ELSE
  THIS^.stSeqCtrlGeneral.eActiveSeqState := E_SEQ_GENERAL.ERROR;
END_CASE
END_METHOD

METHOD PRIVATE _m_Seq_PRESSURE_CALIBRATION : E_SEQ_PROCESS
VAR_INPUT
END_VAR
VAR
	ActiveSeq:  STRING;
END_VAR
//THIS^._m_GeneralStepSetting(StepType:=E_STEP_STATE_TYPE.INIT,
ActiveSeq := TO_STRING(THIS^.eSeq);

CASE THIS^.stSeqCtrlGeneral.eActiveSeqState OF
E_SEQ_GENERAL.READY:;

	
E_SEQ_GENERAL.EXECUTE:;
	IF TRUE
	THEN
		THIS^.stSeqCtrlGeneral.eActiveSeqState := E_SEQ_GENERAL.RESET;
	END_IF
  
E_SEQ_GENERAL.RESET:;
	stSeqCtrlGeneral.iInternalSeqStateCase := 0;
	IF TRUE
	THEN
    THIS^.ii := 1;
    FOR THIS^.ii := 1 TO 7 BY 1 DO
      THIS^.listCalibrationTable[THIS^.ii].uiValue := 0;
      THIS^.listCalibrationTable[THIS^.ii].uiPressure := 0;
      THIS^.listCalibrationTable[THIS^.ii].uiState := 0;
		END_FOR
    THIS^.ii := 1;
		THIS^.stSeqCtrlGeneral.eActiveSeqState := E_SEQ_GENERAL.BUSY;
	END_IF
  
E_SEQ_GENERAL.BUSY:;
	CASE THIS^.stSeqCtrlGeneral.iInternalSeqStateCase OF
		0:	// Set work pressure value to XXXX
      IF TRUE
      AND THIS^.itfValve_PressureLimit.M_SetLimit(ePressureType:= E_PRESSURE_TYPE.VALUE, rLimit:= 1000 * THIS^.ii)
			THEN 
        THIS^.listCalibrationTable[THIS^.ii].uiValue := TO_UINT(1000 * THIS^.ii);
        THIS^.listCalibrationTable[THIS^.ii].uiState := 1;
        THIS^.stSeqCtrlGeneral.iInternalSeqStateCase := 10;
			END_IF
      
    10:	// Set JOG Valve off
      IF TRUE 
      AND THIS^.itfValve_AutomaticEnable.M_ToWP1(tDelay:= T#10MS)
			THEN 
        THIS^.stSeqCtrlGeneral.iInternalSeqStateCase := 20;
			END_IF
      
    20: // Set valves for WP
      IF TRUE
      AND THIS^.itfValve_SinkBlock.M_ToWP1(tDelay:= T#10MS)
      AND THIS^.itfValve_Bypass.M_ToWP1(tDelay:= T#10MS)
      AND THIS^.itfValve_CylCtrl.M_ToWP2(tDelay:= T#10MS)
      THEN
        THIS^.stSeqCtrlGeneral.iInternalSeqStateCase := 30;
			END_IF
      
    30: // Choice step
      IF TRUE
      THEN
        IF THIS^.ii = 1 THEN
          THIS^.stSeqCtrlGeneral.iInternalSeqStateCase := 40;
        ELSE
          THIS^.stSeqCtrlGeneral.iInternalSeqStateCase := 50;
				END_IF
			END_IF
      
    40: // Delay step (wait for cylinder end position)
      IF TRUE
      AND _m_Delay(DelayTime:= T#30S)
      THEN
        THIS^.stSeqCtrlGeneral.iInternalSeqStateCase := 50;
			END_IF
      
    50: // Delay step (cylinder under load)
      IF TRUE
      AND _m_Delay(DelayTime:= T#5S)
      THEN
        THIS^.stSeqCtrlGeneral.iInternalSeqStateCase := 60;
			END_IF
      
    60: // Save pressure
      IF TRUE
      THEN
        THIS^.listCalibrationTable[THIS^.ii].uiPressure := TO_UINT(THIS^.rCurrentPressureInBar);
        THIS^.listCalibrationTable[THIS^.ii].uiState := 2;
        THIS^.stSeqCtrlGeneral.iInternalSeqStateCase := 70;
			END_IF
      
    70: // Decide step
      IF TRUE
      AND _m_Delay(DelayTime:= T#1S)
      THEN
        IF THIS^.ii >= 7 OR THIS^.ii < 1 THEN
          THIS^.ii := 1;
          THIS^.stSeqCtrlGeneral.iInternalSeqStateCase := 1000;
        ELSE
          THIS^.ii := THIS^.ii + 1;
          THIS^.stSeqCtrlGeneral.iInternalSeqStateCase := 0;
				END_IF
			END_IF
      
    1000: // Stop and exit
      IF TRUE
      AND THIS^.itfValve_CylCtrl.M_ToHP(tDelay:= T#10MS)
      AND THIS^.itfValve_Bypass.M_ToHP(tDelay:= T#10MS)
			THEN 
				THIS^.stSeqCtrlGeneral.iInternalSeqStateCase := 9999;
			END_IF
      
	ELSE
		THIS^.stSeqCtrlGeneral.eActiveSeqState := E_SEQ_GENERAL.DONE;  
	END_CASE
	THIS^.stSeqCtrlGeneral.strExtraInfo := CONCAT('Internal state: ', TO_STRING(THIS^.stSeqCtrlGeneral.iInternalSeqStateCase));

E_SEQ_GENERAL.DONE:;

E_SEQ_GENERAL.ERROR:;

E_SEQ_GENERAL.TIME_OUT:; 
IF TRUE
AND THIS^.stSeqCtrlGeneral.bTimeOutActiveQuit 
THEN
  THIS^.stSeqCtrlGeneral.strExtraInfo := 'Bitte quittieren und erneut testen';
  IF TRUE
  //AND itfOpMode.P_QUIT
  THEN
    THIS^.stSeqCtrlGeneral.eActiveSeqState := E_SEQ_GENERAL.EXECUTE;
	END_IF
  
END_IF

ELSE
  THIS^.stSeqCtrlGeneral.eActiveSeqState := E_SEQ_GENERAL.ERROR;
END_CASE
END_METHOD

METHOD PRIVATE _m_Seq_SET_WORK_PRESSURE : E_SEQ_PROCESS
VAR_INPUT
END_VAR
VAR
	ActiveSeq: STRING;
END_VAR
//THIS^._m_GeneralStepSetting(StepType:=E_STEP_STATE_TYPE.INIT,
ActiveSeq := TO_STRING(THIS^.eSeq);

CASE THIS^.stSeqCtrlGeneral.eActiveSeqState OF
E_SEQ_GENERAL.READY:;

	
E_SEQ_GENERAL.EXECUTE:;
	IF TRUE
	THEN
		THIS^.stSeqCtrlGeneral.eActiveSeqState := E_SEQ_GENERAL.RESET;
	END_IF
  
E_SEQ_GENERAL.RESET:;
	stSeqCtrlGeneral.iInternalSeqStateCase := 0;
	IF TRUE
	THEN
		THIS^.stSeqCtrlGeneral.eActiveSeqState := E_SEQ_GENERAL.BUSY;
	END_IF
  
E_SEQ_GENERAL.BUSY:;
	CASE THIS^.stSeqCtrlGeneral.iInternalSeqStateCase OF
		0:	// Set work pressure
      IF TRUE
      AND THIS^.itfValve_PressureLimit.M_SetLimit(ePressureType:= E_PRESSURE_TYPE.VALUE, rLimit:= TO_REAL(THIS^.iTargetPressureAsValueA))
			THEN 
        THIS^.stSeqCtrlGeneral.iInternalSeqStateCase := 1000;
			END_IF
      
    1000: // Exit step
      IF TRUE
			THEN 
				THIS^.stSeqCtrlGeneral.iInternalSeqStateCase := 9999;
			END_IF
      
	ELSE
		THIS^.stSeqCtrlGeneral.eActiveSeqState := E_SEQ_GENERAL.DONE;  
	END_CASE
	THIS^.stSeqCtrlGeneral.strExtraInfo := CONCAT('Internal state: ', TO_STRING(THIS^.stSeqCtrlGeneral.iInternalSeqStateCase));

E_SEQ_GENERAL.DONE:;

E_SEQ_GENERAL.ERROR:;

E_SEQ_GENERAL.TIME_OUT:; 
IF TRUE
AND THIS^.stSeqCtrlGeneral.bTimeOutActiveQuit 
THEN
  THIS^.stSeqCtrlGeneral.strExtraInfo := 'Bitte quittieren und erneut testen';
  IF TRUE
  //AND itfOpMode.P_QUIT
  THEN
    THIS^.stSeqCtrlGeneral.eActiveSeqState := E_SEQ_GENERAL.EXECUTE;
	END_IF
  
END_IF

ELSE
  THIS^.stSeqCtrlGeneral.eActiveSeqState := E_SEQ_GENERAL.ERROR;
END_CASE
END_METHOD

METHOD PRIVATE _m_Seq_STOP : E_SEQ_PROCESS
VAR_INPUT
END_VAR
VAR
	ActiveSeq: STRING;
END_VAR
VAR
	
END_VAR
//THIS^._m_GeneralStepSetting(StepType:=E_STEP_STATE_TYPE.INIT,
ActiveSeq := TO_STRING(THIS^.eSeq);

CASE THIS^.stSeqCtrlGeneral.eActiveSeqState OF
E_SEQ_GENERAL.READY:;

	
E_SEQ_GENERAL.EXECUTE:;
	IF TRUE
	THEN
    THIS^.bRegulationTrigger := FALSE;
		THIS^.stSeqCtrlGeneral.eActiveSeqState := E_SEQ_GENERAL.RESET;
	END_IF
  
E_SEQ_GENERAL.RESET:;
	stSeqCtrlGeneral.iInternalSeqStateCase := 0;
	IF TRUE
	THEN
		THIS^.stSeqCtrlGeneral.eActiveSeqState := E_SEQ_GENERAL.BUSY;
	END_IF
  
E_SEQ_GENERAL.BUSY:;
	CASE THIS^.stSeqCtrlGeneral.iInternalSeqStateCase OF
		0: // Switch off valves
      IF TRUE
      AND THIS^.itfValve_Bypass.M_ToHP(tDelay:= T#0MS)
      AND THIS^.itfValve_CylCtrl.M_ToHP(tDelay:= T#0MS)
			THEN 
				THIS^.stSeqCtrlGeneral.iInternalSeqStateCase := 1000;
			END_IF
      
    1000: // Exit step
      IF TRUE
			THEN 
				THIS^.stSeqCtrlGeneral.iInternalSeqStateCase := 9999;
			END_IF
      
	ELSE
		THIS^.stSeqCtrlGeneral.eActiveSeqState := E_SEQ_GENERAL.DONE;  
	END_CASE
	THIS^.stSeqCtrlGeneral.strExtraInfo := CONCAT('Internal state: ', TO_STRING(THIS^.stSeqCtrlGeneral.iInternalSeqStateCase));

E_SEQ_GENERAL.DONE:;

E_SEQ_GENERAL.ERROR:;

E_SEQ_GENERAL.TIME_OUT:; 
IF TRUE
AND THIS^.stSeqCtrlGeneral.bTimeOutActiveQuit 
THEN
  THIS^.stSeqCtrlGeneral.strExtraInfo := 'Bitte quittieren und erneut testen';
  IF TRUE
  //AND itfOpMode.P_QUIT
  THEN
    THIS^.stSeqCtrlGeneral.eActiveSeqState := E_SEQ_GENERAL.EXECUTE;
	END_IF
  
END_IF

ELSE
  THIS^.stSeqCtrlGeneral.eActiveSeqState := E_SEQ_GENERAL.ERROR;
END_CASE
END_METHOD

METHOD PRIVATE _m_Seq_TO_HP : E_SEQ_PROCESS
VAR_INPUT
END_VAR
VAR
	ActiveSeq: STRING;
END_VAR
VAR
	
END_VAR
//THIS^._m_GeneralStepSetting(StepType:=E_STEP_STATE_TYPE.INIT,
ActiveSeq := TO_STRING(THIS^.eSeq);

CASE THIS^.stSeqCtrlGeneral.eActiveSeqState OF
E_SEQ_GENERAL.READY:;

	
E_SEQ_GENERAL.EXECUTE:;
	IF TRUE
	THEN
    THIS^.bRegulationTrigger := FALSE;
		THIS^.stSeqCtrlGeneral.eActiveSeqState := E_SEQ_GENERAL.RESET;
	END_IF
  
E_SEQ_GENERAL.RESET:;
	stSeqCtrlGeneral.iInternalSeqStateCase := 0;
	IF TRUE
	THEN
		THIS^.stSeqCtrlGeneral.eActiveSeqState := E_SEQ_GENERAL.BUSY;
	END_IF
  
E_SEQ_GENERAL.BUSY:;
	CASE THIS^.stSeqCtrlGeneral.iInternalSeqStateCase OF
		0:	// Set JOG Valve on/off
      IF TRUE 
      AND itfOpMode.P_OP_MODE_STATE = OP_MODE.AUTO
			THEN 
        IF THIS^.itfValve_AutomaticEnable.M_ToWP1(tDelay:= T#0MS) THEN
          THIS^.stSeqCtrlGeneral.iInternalSeqStateCase := 10;
				END_IF
      ELSE
        IF THIS^.itfValve_AutomaticEnable.M_ToHP(tDelay:= T#0MS) THEN
          THIS^.stSeqCtrlGeneral.iInternalSeqStateCase := 10;
				END_IF
			END_IF
      
    10:	// Set work pressure
      IF TRUE
      AND THIS^.itfValve_PressureLimit.M_SetLimit(ePressureType:= E_PRESSURE_TYPE.VALUE, rLimit:= TO_REAL(THIS^.iTargetPressureAsValueB))
			THEN 
        THIS^.stSeqCtrlGeneral.iInternalSeqStateCase := 20;
			END_IF
      
    20: // Set valves
      IF TRUE
      AND THIS^.itfValve_SinkBlock.M_ToWP1(tDelay:= T#0MS)
      AND THIS^.itfValve_Bypass.M_ToWP1(tDelay:= T#0MS)
      AND THIS^.itfValve_CylCtrl.M_ToWP1(tDelay:= T#0MS)
      THEN
        THIS^.stSeqCtrlGeneral.iInternalSeqStateCase := 1000;
			END_IF
      
    1000: // Exit step
      IF TRUE
			THEN 
				THIS^.stSeqCtrlGeneral.iInternalSeqStateCase := 9999;
			END_IF
      
	ELSE
		THIS^.stSeqCtrlGeneral.eActiveSeqState := E_SEQ_GENERAL.DONE;  
	END_CASE
	THIS^.stSeqCtrlGeneral.strExtraInfo := CONCAT('Internal state: ', TO_STRING(THIS^.stSeqCtrlGeneral.iInternalSeqStateCase));

E_SEQ_GENERAL.DONE:;
  THIS^.bRegulationTrigger := THIS^.bRegulation;

E_SEQ_GENERAL.ERROR:;

E_SEQ_GENERAL.TIME_OUT:; 
IF TRUE
AND THIS^.stSeqCtrlGeneral.bTimeOutActiveQuit 
THEN
  THIS^.stSeqCtrlGeneral.strExtraInfo := 'Bitte quittieren und erneut testen';
  IF TRUE
  //AND itfOpMode.P_QUIT
  THEN
    THIS^.stSeqCtrlGeneral.eActiveSeqState := E_SEQ_GENERAL.EXECUTE;
	END_IF
  
END_IF

ELSE
  THIS^.stSeqCtrlGeneral.eActiveSeqState := E_SEQ_GENERAL.ERROR;
END_CASE
END_METHOD

METHOD PRIVATE _m_Seq_TO_WP : E_SEQ_PROCESS
VAR_INPUT
END_VAR
VAR
	ActiveSeq: STRING;
END_VAR
VAR
	
END_VAR
//THIS^._m_GeneralStepSetting(StepType:=E_STEP_STATE_TYPE.INIT,
ActiveSeq := TO_STRING(THIS^.eSeq);

CASE THIS^.stSeqCtrlGeneral.eActiveSeqState OF
E_SEQ_GENERAL.READY:;

	
E_SEQ_GENERAL.EXECUTE:;
	IF TRUE
  //AND _m_Delay(DelayTime:= T#10MS)
	THEN
    THIS^.bRegulationTrigger := FALSE;
		THIS^.stSeqCtrlGeneral.eActiveSeqState := E_SEQ_GENERAL.RESET;
	END_IF
  
E_SEQ_GENERAL.RESET:;
	stSeqCtrlGeneral.iInternalSeqStateCase := 0;
	IF TRUE
	THEN
		THIS^.stSeqCtrlGeneral.eActiveSeqState := E_SEQ_GENERAL.BUSY;
	END_IF
  
E_SEQ_GENERAL.BUSY:;
	CASE THIS^.stSeqCtrlGeneral.iInternalSeqStateCase OF
		0:	// Set JOG Valve on/off
      IF TRUE 
      AND itfOpMode.P_OP_MODE_STATE = OP_MODE.AUTO
			THEN 
        IF THIS^.itfValve_AutomaticEnable.M_ToWP1(tDelay:= T#0MS) THEN
          THIS^.stSeqCtrlGeneral.iInternalSeqStateCase := 10;
				END_IF
      ELSE
        IF THIS^.itfValve_AutomaticEnable.M_ToHP(tDelay:= T#0MS) THEN
          THIS^.stSeqCtrlGeneral.iInternalSeqStateCase := 10;
				END_IF
			END_IF
      
    10:	// Set work pressure
      IF TRUE
      AND THIS^.itfValve_PressureLimit.M_SetLimit(ePressureType:= E_PRESSURE_TYPE.VALUE, rLimit:= TO_REAL(THIS^.iTargetPressureAsValueA))
			THEN 
        THIS^.stSeqCtrlGeneral.iInternalSeqStateCase := 20;
			END_IF
      
    20: // Valves off
      IF TRUE
      AND THIS^.itfValve_SinkBlock.M_ToWP1(tDelay:= T#0MS)
      AND THIS^.itfValve_Bypass.M_ToWP1(tDelay:= T#0MS)
      AND THIS^.itfValve_CylCtrl.M_ToWP2(tDelay:= T#0MS)
      THEN
        THIS^.stSeqCtrlGeneral.iInternalSeqStateCase := 1000;
			END_IF
      
    1000: // Exit step
      IF TRUE
			THEN 
				THIS^.stSeqCtrlGeneral.iInternalSeqStateCase := 9999;
			END_IF
      
	ELSE
		THIS^.stSeqCtrlGeneral.eActiveSeqState := E_SEQ_GENERAL.DONE;  
	END_CASE
	THIS^.stSeqCtrlGeneral.strExtraInfo := CONCAT('Internal state: ', TO_STRING(THIS^.stSeqCtrlGeneral.iInternalSeqStateCase));

E_SEQ_GENERAL.DONE:;
  THIS^.bRegulationTrigger := THIS^.bRegulation;

E_SEQ_GENERAL.ERROR:;

E_SEQ_GENERAL.TIME_OUT:; 
IF TRUE
AND THIS^.stSeqCtrlGeneral.bTimeOutActiveQuit 
THEN
  THIS^.stSeqCtrlGeneral.strExtraInfo := 'Bitte quittieren und erneut testen';
  IF TRUE
  //AND itfOpMode.P_QUIT
  THEN
    THIS^.stSeqCtrlGeneral.eActiveSeqState := E_SEQ_GENERAL.EXECUTE;
	END_IF
  
END_IF

ELSE
  THIS^.stSeqCtrlGeneral.eActiveSeqState := E_SEQ_GENERAL.ERROR;
END_CASE
END_METHOD

METHOD PRIVATE _m_SequenceManager
VAR_INPUT
END_VAR
IF FALSE
//AND THIS^.eActiveSeqState=DONE 
AND eLastSeq<>eSeq
THEN
	IF THIS^.stSeqCtrlGeneral.eActiveSeqState<>E_SEQ_GENERAL.EXECUTE THEN
		THIS^.stSeqCtrlGeneral.eActiveSeqState:=E_SEQ_GENERAL.READY;
	END_IF
END_IF

eSeq := eNextSeq;

//DelayTimer und TimeOut Timer verwalten
stSeqCtrlGeneral.bActiveStep:=	TRUE
				AND eLastSeq					=	eSeq
				AND stSeqCtrlGeneral.eLastActiveSeqState			=	stSeqCtrlGeneral.eActiveSeqState
				AND	stSeqCtrlGeneral.iLastInternalSeqStateCase	=	stSeqCtrlGeneral.iInternalSeqStateCase
				;
			
IF NOT stSeqCtrlGeneral.bActiveStep THEN
	stSeqCtrlGeneral.bDelayActive:=FALSE;
	stSeqCtrlGeneral.bTimeOutActiveQuit:=FALSE;
	stSeqCtrlGeneral.bTimeOutActiveNoQuit:=FALSE;
  THIS^.stSeqCtrlGeneral.strExtraInfo:='';
END_IF

_m_SaveLastStep();
stSeqCtrlGeneral.tonDelay	(IN:=stSeqCtrlGeneral.bActiveStep AND stSeqCtrlGeneral.bDelayActive, 		PT:=stSeqCtrlGeneral.tDelay);
stSeqCtrlGeneral.tonTimeOut	(IN:=stSeqCtrlGeneral.bActiveStep AND (stSeqCtrlGeneral.bTimeOutActiveNoQuit OR stSeqCtrlGeneral.bTimeOutActiveQuit), 	PT:=stSeqCtrlGeneral.tTimeOut);
stSeqCtrlGeneral.tonStepTime	(IN:= stSeqCtrlGeneral.bActiveStep, PT:= T#24H);

IF stSeqCtrlGeneral.tonTimeOut.Q  THEN
	stSeqCtrlGeneral.eActiveSeqState:=E_SEQ_GENERAL.TIME_OUT;
END_IF

IF stSeqCtrlGeneral.iError<>0 THEN
	eSeq:=E_SEQ_CYLINDER.ERROR_SEQ;
END_IF



eLastSeq					:=	eSeq;
stSeqCtrlGeneral.eLastActiveSeqState			:=	stSeqCtrlGeneral.eActiveSeqState;
stSeqCtrlGeneral.iLastInternalSeqStateCase	:=	stSeqCtrlGeneral.iInternalSeqStateCase;

// Reset set ready state
IF THIS^.stSeqCtrlGeneral.bExitSetReadyState THEN
  THIS^.stSeqCtrlGeneral.bExitSetReadyState := FALSE;
END_IF
END_METHOD

METHOD PRIVATE _m_TimeOut : BOOL
VAR_INPUT
	bTimeoutActiveToQuit:	BOOL;
	bTimeOutActiveNoQuit:	BOOL;
	tTimeOut:				TIME;	
END_VAR
THIS^.stSeqCtrlGeneral.bTimeOutActiveQuit:=	bTimeoutActiveToQuit;
THIS^.stSeqCtrlGeneral.bTimeOutActiveNoQuit:=	bTimeOutActiveNoQuit;
THIS^.stSeqCtrlGeneral.tTimeOut:=			tTimeOut;
_m_TimeOut:=FALSE;
IF THIS^.stSeqCtrlGeneral.tonTimeOut.Q THEN
	_m_TimeOut:=TRUE;
END_IF
END_METHOD

METHOD FB_init : BOOL
VAR_INPUT
	bInitRetains : BOOL; // if TRUE, the retain variables are initialized (warm start / cold start)
	bInCopyCode : BOOL;  // if TRUE, the instance afterwards gets moved into the copy code (online change)
  
  itfOpMode:											                        I_OP_MODE; 
  itfEventLogger:                                         I_EVENT_LOGGER;
  itfOpModeVisu:											                    I_OP_MODE_PAUSE_VISU; 
  itfValve_CylCtrl:                                       I_VALVE_X_3;
  itfValve_Bypass:                                        I_VALVE_X_2;
  itfValve_AutomaticEnable:                               I_VALVE_X_2;
  itfValve_SinkBlock:                                     I_VALVE_X_2;
  itfValve_LowPressureCircuitAdd:                         I_VALVE_X_2;
  itfValve_PressureLimit:                                 I_PRV_PROP;
  itfJogBtnPos_Pressed:                                   I_BINARY_SWITCH;
  itfJogBtnNeg_Pressed:                                   I_BINARY_SWITCH;
  lrPistonSurfaceA:                                       LREAL;
  lrPistonSurfaceB:                                       LREAL;
  rEndPosTol:                                             REAL;
  /// Volume flow in l/min or dm³/min
  rPumpVolumeFlow:                                        REAL; // Volumenstrom
  /// Pump efficiency factor (0,5-1)
  rPumpEfficiencyFactor:                                  REAL; // Wirkungsgrad
END_VAR
THIS^.itfOpMode := itfOpMode;
THIS^.itfEventLogger := itfEventLogger;
THIS^.itfOpModeVisu := itfOpModeVisu;
THIS^.itfValve_CylCtrl := itfValve_CylCtrl;
THIS^.itfValve_Bypass := itfValve_Bypass;
THIS^.itfValve_AutomaticEnable := itfValve_AutomaticEnable;
THIS^.itfValve_SinkBlock := itfValve_SinkBlock;
THIS^.itfValve_LowPressureCircuitAdd := itfValve_LowPressureCircuitAdd;
THIS^.itfValve_PressureLimit := itfValve_PressureLimit;
THIS^.itfJogBtnPos_Pressed := itfJogBtnPos_Pressed;
THIS^.itfJogBtnNeg_Pressed := itfJogBtnNeg_Pressed;
THIS^.lrPistonSurfaceA := lrPistonSurfaceA;
THIS^.lrPistonSurfaceB := lrPistonSurfaceB;
THIS^.rEndPosTol := rEndPosTol;
THIS^.rPumpVolumeFlow := rPumpVolumeFlow;
THIS^.rPumpEfficiencyFactor := rPumpEfficiencyFactor;
END_METHOD

METHOD M_AutoMode : BOOL
VAR_INPUT
	bEnable	: BOOL;
END_VAR
END_METHOD

METHOD M_LowPressureCircuit : BOOL
VAR_INPUT
  bAdd:               BOOL;
END_VAR
M_LowPressureCircuit := THIS^.stSeqCtrlGeneral.eActiveSeqState = E_SEQ_GENERAL.DONE;

// Assign input
THIS^.bLowPressureCircuitEnabled := bAdd;

// General
IF THIS^.stSeqCtrlGeneral.eActiveSeqState = E_SEQ_GENERAL.READY THEN
  THIS^.eNextSeq := E_SEQ_CYLINDER.LOW_PRESSURE_CIRCUIT;
  THIS^.stSeqCtrlGeneral.eActiveSeqState := E_SEQ_GENERAL.EXECUTE;
END_IF
END_METHOD

METHOD M_PressureCalibration : BOOL
M_PressureCalibration := THIS^.stSeqCtrlGeneral.eActiveSeqState = E_SEQ_GENERAL.DONE;

// Assign input

// General
IF THIS^.stSeqCtrlGeneral.eActiveSeqState = E_SEQ_GENERAL.READY THEN
  THIS^.eNextSeq := E_SEQ_CYLINDER.PRESSURE_CALIBRATION;
  THIS^.stSeqCtrlGeneral.eActiveSeqState := E_SEQ_GENERAL.EXECUTE;
END_IF
END_METHOD

METHOD M_Reset : BOOL
M_Reset := THIS^.stSeqCtrlGeneral.eActiveSeqState = E_SEQ_GENERAL.DONE;

// General
IF THIS^.stSeqCtrlGeneral.eActiveSeqState = E_SEQ_GENERAL.READY THEN
  THIS^.eNextSeq := E_SEQ_CYLINDER.INIT;
  THIS^.stSeqCtrlGeneral.eActiveSeqState := E_SEQ_GENERAL.EXECUTE;
END_IF
END_METHOD

{warning 'Methodenimplementierung hinzufügen'}
(*=== Method: M_Run  ============================================

 @brief: Here is the global code (Timer, Event, Flange,...)*)
METHOD M_Run
END_METHOD

METHOD M_SetReady : BOOL
VAR_INPUT
END_VAR
M_SetReady := TRUE
              AND THIS^.stSeqCtrlGeneral.eActiveSeqState = E_SEQ_GENERAL.READY
              AND THIS^.eSeq = E_SEQ_CYLINDER.BASE;

THIS^.stSeqCtrlGeneral.eActiveSeqState := E_SEQ_GENERAL.READY;
THIS^.eNextSeq := E_SEQ_CYLINDER.BASE;
END_METHOD

METHOD M_SetWorkPressure : BOOL
VAR_INPUT
  /// Bar | Force in N | Percent 0-100 | Value 0-32767
  ePressureType:                   E_PRESSURE_TYPE;
  rWorkPressure:                   REAL;
END_VAR
M_SetWorkPressure := THIS^.stSeqCtrlGeneral.eActiveSeqState = E_SEQ_GENERAL.DONE;

// Assign input
IF ePressureType = E_PRESSURE_TYPE.BAR THEN
  THIS^.rTargetPressureInBarA := THIS^.rTargetPressureInBarB := rWorkPressure;
  THIS^.rTargetPressureInForceA := rWorkPressure / 10 * THIS^.lrPistonSurfaceA;
  THIS^.rTargetPressureInForceB := rWorkPressure / 10 * THIS^.lrPistonSurfaceB;
  THIS^.rTargetPressureInPercentA := THIS^.rTargetPressureInPercentB := 100 / THIS^.itfValve_PressureLimit.P_MaxLimitInBar * rWorkPressure;
  THIS^.iTargetPressureAsValueA := THIS^.iTargetPressureAsValueB := TO_INT(F_InterpolLinear(lrValueUnscale := rWorkPressure , arrCalibrate:= listCylCalibration, iPts:= 7));
ELSIF ePressureType = E_PRESSURE_TYPE.FORCE THEN
  THIS^.rTargetPressureInForceA := THIS^.rTargetPressureInForceB := rWorkPressure;;
  THIS^.rTargetPressureInBarA := THIS^.rTargetPressureInForceA / THIS^.lrPistonSurfaceA * 10;
  THIS^.rTargetPressureInBarB := THIS^.rTargetPressureInForceB / THIS^.lrPistonSurfaceB * 10;
  THIS^.rTargetPressureInPercentA := 100 / THIS^.itfValve_PressureLimit.P_MaxLimitInBar * THIS^.rTargetPressureInBarA;
  THIS^.rTargetPressureInPercentB := 100 / THIS^.itfValve_PressureLimit.P_MaxLimitInBar * THIS^.rTargetPressureInBarB;
  THIS^.iTargetPressureAsValueA := TO_INT(F_InterpolLinear(lrValueUnscale := THIS^.rTargetPressureInBarA , arrCalibrate:= listCylCalibration, iPts:= 7));
  THIS^.iTargetPressureAsValueB := TO_INT(F_InterpolLinear(lrValueUnscale := THIS^.rTargetPressureInBarB , arrCalibrate:= listCylCalibration, iPts:= 7));
ELSIF ePressureType = E_PRESSURE_TYPE.PERCENT THEN
  THIS^.rTargetPressureInPercentA := THIS^.rTargetPressureInPercentB := rWorkPressure;
  THIS^.rTargetPressureInBarA := THIS^.rTargetPressureInBarB := THIS^.itfValve_PressureLimit.P_MaxLimitInBar / 100 * rWorkPressure;
  THIS^.rTargetPressureInForceA := THIS^.rTargetPressureInBarA / 10 * THIS^.lrPistonSurfaceA;
  THIS^.rTargetPressureInForceB := THIS^.rTargetPressureInBarB / 10 * THIS^.lrPistonSurfaceB;
  THIS^.iTargetPressureAsValueA := TO_INT(F_InterpolLinear(lrValueUnscale := THIS^.rTargetPressureInBarA , arrCalibrate:= listCylCalibration, iPts:= 7));
  THIS^.iTargetPressureAsValueB := TO_INT(F_InterpolLinear(lrValueUnscale := THIS^.rTargetPressureInBarB , arrCalibrate:= listCylCalibration, iPts:= 7));
ELSE
  THIS^.iTargetPressureAsValueA := THIS^.iTargetPressureAsValueB := TO_INT(rWorkPressure);
END_IF

// General
IF THIS^.stSeqCtrlGeneral.eActiveSeqState = E_SEQ_GENERAL.READY THEN
  THIS^.eNextSeq := E_SEQ_CYLINDER.SET_WORK_PRESSURE;
  THIS^.stSeqCtrlGeneral.eActiveSeqState := E_SEQ_GENERAL.EXECUTE;
END_IF
END_METHOD

METHOD M_SetWorkPressureZero : BOOL
M_SetWorkPressureZero := THIS^.stSeqCtrlGeneral.eActiveSeqState = E_SEQ_GENERAL.DONE;

THIS^.iTargetPressureAsValueA := 0;

// General
IF THIS^.stSeqCtrlGeneral.eActiveSeqState = E_SEQ_GENERAL.READY THEN
  THIS^.eNextSeq := E_SEQ_CYLINDER.SET_WORK_PRESSURE;
  THIS^.stSeqCtrlGeneral.eActiveSeqState := E_SEQ_GENERAL.EXECUTE;
END_IF
END_METHOD

METHOD M_Stop : BOOL
M_Stop := THIS^.stSeqCtrlGeneral.eActiveSeqState = E_SEQ_GENERAL.DONE;

// Assign input
THIS^.bRegulation := FALSE;
THIS^.rActiveForce := 0;
THIS^.iCorrectedPressureAsValue := 0;
THIS^.bRegulationTrigger := FALSE;
THIS^.bRegulationBusy := FALSE;
THIS^.bCorrectionTrigger := FALSE;

// General
IF THIS^.stSeqCtrlGeneral.eActiveSeqState = E_SEQ_GENERAL.READY THEN
  THIS^.eNextSeq := E_SEQ_CYLINDER.STOP;
  THIS^.stSeqCtrlGeneral.eActiveSeqState := E_SEQ_GENERAL.EXECUTE;
END_IF
END_METHOD

METHOD M_ToHP : BOOL
VAR_INPUT
  /// Bar | Force in N | Percent 0-100 | Value 0-32767
  ePressureType:            E_PRESSURE_TYPE;
  rWorkPressure:            REAL;
  bPressureRegulation:      BOOL;
  /// Just need for prop valve
  eSpeedType:               E_SPEED_TYPE;
  rSpeed:                   REAL; 
END_VAR
M_ToHP := THIS^.stSeqCtrlGeneral.eActiveSeqState = E_SEQ_GENERAL.DONE;

// Assign input
IF ePressureType = E_PRESSURE_TYPE.BAR THEN
  THIS^.rTargetPressureInBarA := THIS^.rTargetPressureInBarB := rWorkPressure;
  THIS^.rTargetPressureInForceA := rWorkPressure / 10 * THIS^.lrPistonSurfaceA;
  THIS^.rTargetPressureInForceB := rWorkPressure / 10 * THIS^.lrPistonSurfaceB;
  THIS^.rTargetPressureInPercentA := THIS^.rTargetPressureInPercentB := 100 / THIS^.itfValve_PressureLimit.P_MaxLimitInBar * rWorkPressure;
  THIS^.iTargetPressureAsValueA := THIS^.iTargetPressureAsValueB := THIS^.iCorrectedPressureAsValue := TO_INT(F_InterpolLinear(lrValueUnscale := rWorkPressure , arrCalibrate:= listCylCalibration, iPts:= 7));
ELSIF ePressureType = E_PRESSURE_TYPE.FORCE THEN
  THIS^.rTargetPressureInForceA := THIS^.rTargetPressureInForceB := rWorkPressure;;
  THIS^.rTargetPressureInBarA := THIS^.rTargetPressureInForceA / THIS^.lrPistonSurfaceA * 10;
  THIS^.rTargetPressureInBarB := THIS^.rTargetPressureInForceB / THIS^.lrPistonSurfaceB * 10;
  THIS^.rTargetPressureInPercentA := 100 / THIS^.itfValve_PressureLimit.P_MaxLimitInBar * THIS^.rTargetPressureInBarA;
  THIS^.rTargetPressureInPercentB := 100 / THIS^.itfValve_PressureLimit.P_MaxLimitInBar * THIS^.rTargetPressureInBarB;
  THIS^.iTargetPressureAsValueA := THIS^.iCorrectedPressureAsValue := TO_INT(F_InterpolLinear(lrValueUnscale := THIS^.rTargetPressureInBarA , arrCalibrate:= listCylCalibration, iPts:= 7));
  THIS^.iTargetPressureAsValueB := TO_INT(F_InterpolLinear(lrValueUnscale := THIS^.rTargetPressureInBarB , arrCalibrate:= listCylCalibration, iPts:= 7));
ELSIF ePressureType = E_PRESSURE_TYPE.PERCENT THEN
  THIS^.rTargetPressureInPercentA := THIS^.rTargetPressureInPercentB := rWorkPressure;
  THIS^.rTargetPressureInBarA := THIS^.rTargetPressureInBarB := THIS^.itfValve_PressureLimit.P_MaxLimitInBar / 100 * rWorkPressure;
  THIS^.rTargetPressureInForceA := THIS^.rTargetPressureInBarA / 10 * THIS^.lrPistonSurfaceA;
  THIS^.rTargetPressureInForceB := THIS^.rTargetPressureInBarB / 10 * THIS^.lrPistonSurfaceB;
  THIS^.iTargetPressureAsValueA := THIS^.iCorrectedPressureAsValue := TO_INT(F_InterpolLinear(lrValueUnscale := THIS^.rTargetPressureInBarA , arrCalibrate:= listCylCalibration, iPts:= 7));
  THIS^.iTargetPressureAsValueB := TO_INT(F_InterpolLinear(lrValueUnscale := THIS^.rTargetPressureInBarB , arrCalibrate:= listCylCalibration, iPts:= 7));
ELSE
  THIS^.iTargetPressureAsValueA := THIS^.iTargetPressureAsValueB := THIS^.iCorrectedPressureAsValue := TO_INT(rWorkPressure);
END_IF
THIS^.bRegulation := bPressureRegulation;

// General
IF THIS^.stSeqCtrlGeneral.eActiveSeqState = E_SEQ_GENERAL.READY THEN
  THIS^.eNextSeq := E_SEQ_CYLINDER.TO_HP;
  THIS^.stSeqCtrlGeneral.eActiveSeqState := E_SEQ_GENERAL.EXECUTE;
END_IF
END_METHOD

METHOD M_ToWP : BOOL
VAR_INPUT
  /// Bar | Force in N | Percent 0-100 | Value 0-32767
  ePressureType:            E_PRESSURE_TYPE;
  rWorkPressure:            REAL;
  bPressureRegulation:      BOOL;
  /// Just need for prop valve
  eSpeedType:               E_SPEED_TYPE;
  rSpeed:                   REAL; 
END_VAR
M_ToWP := THIS^.stSeqCtrlGeneral.eActiveSeqState = E_SEQ_GENERAL.DONE;

// Assign input
IF ePressureType = E_PRESSURE_TYPE.BAR THEN
  THIS^.rTargetPressureInBarA := THIS^.rTargetPressureInBarB := rWorkPressure;
  THIS^.rTargetPressureInForceA := rWorkPressure / 10 * THIS^.lrPistonSurfaceA;
  THIS^.rTargetPressureInForceB := rWorkPressure / 10 * THIS^.lrPistonSurfaceB;
  THIS^.rTargetPressureInPercentA := THIS^.rTargetPressureInPercentB := 100 / THIS^.itfValve_PressureLimit.P_MaxLimitInBar * rWorkPressure;
  THIS^.iTargetPressureAsValueA := THIS^.iTargetPressureAsValueB := THIS^.iCorrectedPressureAsValue := TO_INT(F_InterpolLinear(lrValueUnscale := rWorkPressure , arrCalibrate:= listCylCalibration, iPts:= 7));
ELSIF ePressureType = E_PRESSURE_TYPE.FORCE THEN
  THIS^.rTargetPressureInForceA := THIS^.rTargetPressureInForceB := rWorkPressure;;
  THIS^.rTargetPressureInBarA := THIS^.rTargetPressureInForceA / THIS^.lrPistonSurfaceA * 10;
  THIS^.rTargetPressureInBarB := THIS^.rTargetPressureInForceB / THIS^.lrPistonSurfaceB * 10;
  THIS^.rTargetPressureInPercentA := 100 / THIS^.itfValve_PressureLimit.P_MaxLimitInBar * THIS^.rTargetPressureInBarA;
  THIS^.rTargetPressureInPercentB := 100 / THIS^.itfValve_PressureLimit.P_MaxLimitInBar * THIS^.rTargetPressureInBarB;
  THIS^.iTargetPressureAsValueA := THIS^.iCorrectedPressureAsValue := TO_INT(F_InterpolLinear(lrValueUnscale := THIS^.rTargetPressureInBarA , arrCalibrate:= listCylCalibration, iPts:= 7));
  THIS^.iTargetPressureAsValueB := TO_INT(F_InterpolLinear(lrValueUnscale := THIS^.rTargetPressureInBarB , arrCalibrate:= listCylCalibration, iPts:= 7));
ELSIF ePressureType = E_PRESSURE_TYPE.PERCENT THEN
  THIS^.rTargetPressureInPercentA := THIS^.rTargetPressureInPercentB := rWorkPressure;
  THIS^.rTargetPressureInBarA := THIS^.rTargetPressureInBarB := THIS^.itfValve_PressureLimit.P_MaxLimitInBar / 100 * rWorkPressure;
  THIS^.rTargetPressureInForceA := THIS^.rTargetPressureInBarA / 10 * THIS^.lrPistonSurfaceA;
  THIS^.rTargetPressureInForceB := THIS^.rTargetPressureInBarB / 10 * THIS^.lrPistonSurfaceB;
  THIS^.iTargetPressureAsValueA := THIS^.iCorrectedPressureAsValue := TO_INT(F_InterpolLinear(lrValueUnscale := THIS^.rTargetPressureInBarA , arrCalibrate:= listCylCalibration, iPts:= 7));
  THIS^.iTargetPressureAsValueB := TO_INT(F_InterpolLinear(lrValueUnscale := THIS^.rTargetPressureInBarB , arrCalibrate:= listCylCalibration, iPts:= 7));
ELSE
  THIS^.iTargetPressureAsValueA := THIS^.iTargetPressureAsValueB := THIS^.iCorrectedPressureAsValue := TO_INT(rWorkPressure);
END_IF
THIS^.bRegulation := bPressureRegulation;

// General
IF THIS^.stSeqCtrlGeneral.eActiveSeqState = E_SEQ_GENERAL.READY THEN
  THIS^.eNextSeq := E_SEQ_CYLINDER.TO_WP;
  THIS^.stSeqCtrlGeneral.eActiveSeqState := E_SEQ_GENERAL.EXECUTE;
END_IF
END_METHOD

{warning 'Eigenschaftenimplementierung hinzufügen'}
PROPERTY P_CurrentForceInKN : REAL
GET
IF THIS^.itfValve_CylCtrl.P_InWP2 THEN
  P_CurrentForceInKN := THIS^.rCurrentPressureInBar / 10000 * THIS^.lrPistonSurfaceA;
  THIS^.rActiveForce := THIS^.rTargetPressureInForceA;
ELSIF THIS^.itfValve_CylCtrl.P_InWP1 THEN
  P_CurrentForceInKN := THIS^.rCurrentPressureInBar / 10000 * THIS^.lrPistonSurfaceB;
  THIS^.rActiveForce := THIS^.rTargetPressureInForceB;
ELSE
  P_CurrentForceInKN := 0;
END_IF
END_GET
END_PROPERTY

{warning 'Eigenschaftenimplementierung hinzufügen'}
(*=== Property: P_Event  ============================================

 @param [set]: 	Set the Structure "ST_EVENT" from another Object
 @param [get]: 	Return the Structure "ST_EVENT", it contains the actual 
					event of the Object *)
PROPERTY P_Event : GenLib.ST_EVENT
GET
END_GET
SET
END_SET
END_PROPERTY

{warning 'Eigenschaftenimplementierung hinzufügen'}
(*=== Property: P_FullObjectPath  ============================================

 @param [set]: 	Set the Object Path (Clear String of Object)
 @param [get]: 	Return the Objectpath *)
PROPERTY P_FullObjectPath : STRING
GET
P_FullObjectPath := strInstancePath;
END_GET
SET
strInstancePath := P_FullObjectPath;
END_SET
END_PROPERTY

{warning 'Eigenschaftenimplementierung hinzufügen'}
(*=== Property: P_Global_Ack  ============================================

 @param [set]: 	Set the Bit for Ack from another Object
 @param [get]: 	Return the state of Ack Bit*)
PROPERTY P_Global_Ack : BOOL
GET
END_GET
SET
END_SET
END_PROPERTY

{warning 'Eigenschaftenimplementierung hinzufügen'}
(*=== Property: P_GlobalID  ============================================

 @param [set]: 	-
 @param [get]: 	Return the string of instance path*)
PROPERTY P_GlobalID : STRING
GET
END_GET
END_PROPERTY

{warning 'Eigenschaftenimplementierung hinzufügen'}
PROPERTY P_PistonSurfaceA : LREAL
GET
P_PistonSurfaceA := THIS^.lrPistonSurfaceA;
END_GET
END_PROPERTY

{warning 'Eigenschaftenimplementierung hinzufügen'}
PROPERTY P_PistonSurfaceB : LREAL
GET
P_PistonSurfaceB := THIS^.lrPistonSurfaceB;
END_GET
END_PROPERTY

{warning 'Eigenschaftenimplementierung hinzufügen'}
PROPERTY P_PressureOk : BOOL
GET
END_GET
END_PROPERTY

{warning 'Eigenschaftenimplementierung hinzufügen'}
PROPERTY P_ReadyState : BOOL
GET
P_ReadyState := THIS^.stSeqCtrlGeneral.eActiveSeqState = E_SEQ_GENERAL.READY;
END_GET
END_PROPERTY

PROPERTY P_WorkPressure : REAL
GET
P_WorkPressure := THIS^.rCurrentPressureInBar;
END_GET
END_PROPERTY

END_FUNCTION_BLOCK

// ---- PROGRAMS/PrgVisu.TcPOU
{attribute 'global_init_slot' := '40030'}
PROGRAM PrgVisu
VAR
	fbVisuOPMode:						                        FB_OP_MODE_PAUSE_VISU(itfOpMode:= PrgOrg.fbOpMode);
  tonHeartbeat:                                   TON;
  
  bInit : 									                      BOOL; 
  bSend : 									                      BOOL; 
  fbMsg : 									                      FB_TcMessage;
  fbAlarm:                                        FB_TcAlarm;
  bMachineLightOn:                                BOOL := TRUE;
  fbEventLogger:                                  FB_EVENT_LOGGER();
END_VAR
VAR //HMI enables
  fbHMICtrl:                                      FB_HMI_CTRL_ADS(itfOpMode:= PrgOrg.fbOpMode,
                                                                  itfEventLogger:= PrgOrg.fbEventLogger);
  bEnableAuto:                                    BOOL;
  bEnableEnduranceRun:                            BOOL;
  bEnableLeakTest1:                               BOOL;
  bEnableLeakTest2:                               BOOL;
  bEnableBreakPressureDet:                        BOOL;
  bEnableManual:                                  BOOL;
  bEnableHand:                                    BOOL;
  bEnableJog:                                     BOOL;
  bEnableInit:                                    BOOL;
  bEnableDoorLock:                                BOOL;
  bEnableAck:                                     BOOL;
  bEnableParams:                                  BOOL;
  bEnableOptions:                                 BOOL;
  bEnableSelection:                               BOOL;
  bPumpsOn:                                       BOOL;
END_VAR
VAR
  uiHMISeq:                                       UINT := 0;
  bStartHMI:                                      BOOL;
  bCloseHMI:                                      BOOL;
  bOpenKeyboard:                                  BOOL;
  bHideKeyboard:                                  BOOL;
  bShutdownPc:                                    BOOL;
  bRestartPc:                                     BOOL;
  liFreeSpaceOnC:                                 LINT;
END_VAR
VAR // Parameter: Selected ComboBox Index
  uiCmbCylinder:                                  UINT := 0;
  uiCmbEnduranceRun:                              UINT := 0;
  uiCmbGeneralSettings:                           UINT := 0;
  uiCmbLeakTest1:                                 UINT := 0;
  uiCmbLeakTest2:                                 UINT := 0;
  uiCmbBreakPressureDet:                          UINT := 0;
END_VAR

(* Actions *)
A_000_FBs();
A_010_Init();
A_020_Enables();
A_030_HMIControl();

ACTION A_000_FBs:
(* FBs *)
fbVisuOPMode();
fbHMICtrl(bLifeBit:= PrgMeasure.bLifeBit,
          bAdsConnected:= PrgMeasure.bAdsConnected,
          bReady:= PrgMeasure.bReady,
          bBusy:= PrgMeasure.bBusy,
          liFreeSpaceOnC=> liFreeSpaceOnC);
END_ACTION

ACTION A_010_Init:
tonHeartbeat(in:=NOT tonHeartbeat.Q, pt:=T#100MS);
END_ACTION

ACTION A_020_Enables:
(* Enables *)
bPumpsOn := TRUE
            AND PrgStation.fbBypassPump.P_State
            AND PrgStation.fbCounterCyl1Pump.P_State
            AND PrgStation.fbCounterCyl2Pump.P_State
            AND PrgStation.fbCounterCyl3Pump.P_State
            AND PrgStation.fbCounterCyl4Pump.P_State
            AND PrgStation.fbLowPressurePump.P_State
            AND PrgStation.fbOilCooler.P_State
            AND PrgStation.fbTestCyl1Pump.P_State
            AND PrgStation.fbTestCyl2Pump.P_State
            AND PrgStation.fbTestCyl3Pump.P_State
            AND PrgStation.fbTestCyl4Pump.P_State;
            
bEnableAuto := TRUE
               AND (bEnableEnduranceRun
                 OR bEnableLeakTest1
                 OR bEnableLeakTest2
                 OR bEnableBreakPressureDet);

bEnableEnduranceRun := TRUE
               AND (NOT (fbVisuOPMode.b_Automatic OR fbVisuOPMode.b_Manual OR fbVisuOPMode.b_Reset)
               AND PrgOrg.bInitOK
               AND ((PrgStation.fbNest1.bEnable AND PrgStation.sTestCyl1SNo<>'') 
                 OR (PrgStation.fbNest2.bEnable AND PrgStation.sTestCyl2SNo<>'') 
                 OR (PrgStation.fbNest3.bEnable AND PrgStation.sTestCyl2SNo<>'')
                 OR (PrgStation.fbNest4.bEnable AND PrgStation.sTestCyl2SNo<>''))
               AND NOT PrgOrg.fbOpMode.P_EMERGANCY_STOP
               AND bPumpsOn
               AND PrgOrg.fbFromSafety_SafetyDoor_Ok.P_Active);
               
bEnableLeakTest1 := TRUE
                    AND (NOT (fbVisuOPMode.b_Automatic OR fbVisuOPMode.b_Manual OR fbVisuOPMode.b_Reset)
                    AND PrgOrg.bInitOK
                    AND ((PrgStation.fbNest1.bEnable AND PrgStation.sTestCyl1SNo<>'') 
                      OR (PrgStation.fbNest2.bEnable AND PrgStation.sTestCyl2SNo<>'') 
                      OR (PrgStation.fbNest3.bEnable AND PrgStation.sTestCyl2SNo<>'')
                      OR (PrgStation.fbNest4.bEnable AND PrgStation.sTestCyl2SNo<>''))
                    AND NOT PrgOrg.fbOpMode.P_EMERGANCY_STOP
                    AND bPumpsOn
                    AND PrgOrg.fbFromSafety_SafetyDoor_Ok.P_Active);
                    
bEnableLeakTest2 := TRUE
                    AND (NOT (fbVisuOPMode.b_Automatic OR fbVisuOPMode.b_Manual OR fbVisuOPMode.b_Reset)
                    AND PrgOrg.bInitOK
                    AND (PrgStation.fbNest1.bEnable AND PrgStation.sTestCyl1SNo<>'')
                    AND NOT PrgOrg.fbOpMode.P_EMERGANCY_STOP
                    AND bPumpsOn
                    AND PrgOrg.fbFromSafety_SafetyDoor_Ok.P_Active);
                    
bEnableBreakPressureDet := TRUE
                           AND (NOT (fbVisuOPMode.b_Automatic OR fbVisuOPMode.b_Manual OR fbVisuOPMode.b_Reset)
                           AND PrgOrg.bInitOK
                           AND (PrgStation.fbNest1.bEnable AND PrgStation.sTestCyl1SNo<>'')
                           AND NOT PrgOrg.fbOpMode.P_EMERGANCY_STOP
                           AND bPumpsOn
                           AND PrgOrg.fbFromSafety_SafetyDoor_Ok.P_Active);
               
bEnableManual := TRUE
                 AND (bEnableHand
                   OR bEnableJog);
               
bEnableHand := TRUE
               AND (NOT (fbVisuOPMode.b_Automatic 
                 OR fbVisuOPMode.b_Manual 
                 OR fbVisuOPMode.b_Reset) 
               AND bPumpsOn
               AND PrgOrg.fbFromSafety_SafetyDoor_Ok.P_Active);
                 
bEnableJog := TRUE
              AND (NOT (fbVisuOPMode.b_Automatic 
                OR fbVisuOPMode.b_Manual 
                OR fbVisuOPMode.b_Reset) 
              AND bPumpsOn);
                 
bEnableInit := TRUE
               AND (NOT (fbVisuOPMode.b_Automatic 
                 OR fbVisuOPMode.b_Manual 
                 OR fbVisuOPMode.b_Reset 
                 OR PrgStation.bBusyInit)
               AND PrgOrg.fbFromSafety_SafetyDoor_Ok.P_Active);
                 
bEnableDoorLock := TRUE
                   AND (NOT (fbVisuOPMode.b_Automatic 
                     OR fbVisuOPMode.b_Reset) 
                   OR PrgStation.fbMainProcess.bShowMessage);
                   
bEnableAck := TRUE
              AND (NOT (fbVisuOPMode.b_Automatic 
                OR fbVisuOPMode.b_Reset));
                
bEnableParams := TRUE
                 AND PrgOrg.fbOpMode.P_OP_MODE_STATE = OP_MODE.AUTO_TEMPORARY;
                 
bEnableSelection := TRUE
                    AND NOT fbVisuOPMode.b_Automatic;
                 
bEnableOptions := TRUE
                  AND (NOT (fbVisuOPMode.b_Automatic 
                   OR fbVisuOPMode.b_Reset));
END_ACTION

ACTION A_030_HMIControl:
(* HMI control *)
CASE uiHMISeq OF
  0:
    IF fbHMICtrl.M_SetReady() THEN
      IF bStartHMI THEN
        uiHMISeq := 1;
      ELSIF bCloseHMI THEN
        uiHMISeq := 2;
      ELSIF bOpenKeyboard THEN
        uiHMISeq := 3;
      ELSIF bHideKeyboard THEN
        uiHMISeq := 4;
      ELSIF bShutdownPc THEN
        uiHMISeq := 5;
      ELSIF bRestartPc THEN
        uiHMISeq := 6;
			END_IF
		END_IF
  1:
    IF fbHMICtrl.M_StartHMI() THEN
      bStartHMI := FALSE;
      uiHMISeq := 0;
		END_IF
  2:
    IF fbHMICtrl.M_CloseHMI() THEN
      bCloseHMI := FALSE;
      uiHMISeq := 0;
		END_IF
  3:
    IF fbHMICtrl.M_ShowWinKeyboard() THEN
      bOpenKeyboard := FALSE;
      uiHMISeq := 0;
		END_IF
  4:
    IF fbHMICtrl.M_HideWinKeyboard() THEN
      bHideKeyboard := FALSE;
      uiHMISeq := 0;
		END_IF
  5:
    IF fbHMICtrl.M_PCShutdown() THEN
      bShutdownPc := FALSE;
      uiHMISeq := 0;
		END_IF
  6:
    IF fbHMICtrl.M_PCReboot() THEN
      bRestartPc := FALSE;
      uiHMISeq := 0;
		END_IF
END_CASE
END_ACTION

END_PROGRAM

// ---- ORGANISATION/OP_MODE/POU/FB_OP_MODE_PAUSE_VISU.TcPOU
FUNCTION_BLOCK FB_OP_MODE_PAUSE_VISU IMPLEMENTS I_OP_MODE_PAUSE_VISU
VAR
	itfOpMode:                          I_OP_MODE_PAUSE;
	//Press 
	bClick_Automatic:                   BOOL;
	bClick_Debug:                       BOOL;
	bClick_Manual:                      BOOL;
	bClick_Reset:                       BOOL;
	bClick_Start:                       BOOL;
	bClick_Stop:                        BOOL;
	bClick_Pause:                       BOOL;
	//State
	b_Automatic:                        BOOL;
	b_Debug:                            BOOL;
	b_Manual:                           BOOL;
	b_Reset:                            BOOL;
	//temporay State
	btemporay_Automatic:                BOOL;
	btemporay_Debug:                    BOOL;
	btemporay_Manual:                   BOOL;
	btemporay_Reset:                    BOOL;
	iOPModeState:                       INT;
  // Control buttons clicked
  bEnduranceRunClicked:               BOOL;
  bLeakTest1Clicked:                  BOOL;
  bLeakTest2Clicked:                  BOOL;
  bBreakTestClicked:                  BOOL;
  bJogClicked:                        BOOL;
  bHandClicked:                       BOOL;
  bEnduranceRunMode:                  BOOL;
  bLeakTest1Mode:                     BOOL;
  bLeakTest2Mode:                     BOOL;
  bBreakTestMode:                     BOOL;
  bJogMode:                           BOOL;
  bHandMode:                          BOOL;
  
  // JOG Direction
  bJogCounterCyl1_Clicked:            BOOL;
  bJogCounterCyl2_Clicked:            BOOL;
  bJogCounterCyl3_Clicked:            BOOL;
  bJogCounterCyl4_Clicked:            BOOL;
  bJogCounterCyl1_Active:             BOOL;
  bJogCounterCyl2_Active:             BOOL;
  bJogCounterCyl3_Active:             BOOL;
  bJogCounterCyl4_Active:             BOOL;
	fbBlink:                            FB_Blink;
END_VAR
VAR_IN_OUT

END_VAR
VAR
END_VAR


//CLICK to OP-Mode
IF bClick_Automatic	THEN
	itfOpMode.M_AUTOMATIC();
	bClick_Automatic := FALSE;
END_IF
	
IF bClick_Debug	THEN
	itfOpMode.M_DEBUG();
	bClick_Debug := FALSE;
END_IF
		
IF bClick_Manual THEN
	itfOpMode.M_MANUAL();
	bClick_Manual		:= FALSE;
END_IF
			
IF bClick_Reset	THEN
	itfOpMode.M_RESET();
	bClick_Reset		:= FALSE;
  //M_ResetModeSelection();
END_IF
	
		
IF bClick_Start	THEN
	itfOpMode.M_OP_MODE_ON();
	bClick_Start := FALSE;
END_IF
		
IF bClick_Stop THEN
	itfOpMode.M_OP_MODE_OFF();
  //itfOpMode.M_STOP();
	bClick_Stop			:= FALSE;
  //M_ResetModeSelection();
END_IF

IF bClick_Pause	THEN
	itfOpMode.M_OP_MODE_TO_PAUSE();
	bClick_Pause := FALSE;
END_IF
//
b_Automatic := FALSE;
b_Debug := FALSE; 
b_Manual := FALSE;
b_Reset := FALSE;
btemporay_Automatic := FALSE;
btemporay_Debug := FALSE;
btemporay_Manual := FALSE;
btemporay_Reset := FALSE;

//GET OP MODE STATE
CASE itfOpMode.P_OP_MODE_STATE OF		
	OP_MODE.AUTO: 				    b_Automatic := TRUE;
	OP_MODE.PAUSE:				    b_Automatic :=fbBlink.P_1Hz;		
 	OP_MODE.DEBUG:				    b_Debug := TRUE;
	OP_MODE.MANUAL:				    b_Manual := TRUE;
	OP_MODE.INIT:				      b_Reset := fbBlink.P_1Hz;
	OP_MODE.INIT_OK:			    b_Reset := TRUE;							
	OP_MODE.AUTO_TEMPORARY:		btemporay_Automatic := TRUE;
	OP_MODE.DEBUG_TEMPORARY:	btemporay_Debug := TRUE;
	OP_MODE.MANUAL_TEMPORARY:	btemporay_Manual := TRUE;
	OP_MODE.RESET_TEMPORARY:	btemporay_Reset := TRUE;
END_CASE
iOPModeState := itfOpMode.P_OP_MODE_STATE;

// Control buttons clicked
IF bEnduranceRunClicked THEN
  bEnduranceRunClicked := FALSE;
  bEnduranceRunMode := TRUE;
  bLeakTest1Mode := FALSE;
  bLeakTest2Mode := FALSE;
  bBreakTestMode := FALSE;
  bJogMode := FALSE;
  bHandMode := FALSE;
ELSIF bLeakTest1Clicked THEN
  bLeakTest1Clicked := FALSE;
  bEnduranceRunMode := FALSE;
  bLeakTest1Mode := TRUE;
  bLeakTest2Mode := FALSE;
  bBreakTestMode := FALSE;
  bJogMode := FALSE;
  bHandMode := FALSE;
ELSIF bLeakTest2Clicked THEN
  bLeakTest2Clicked := FALSE;
  bEnduranceRunMode := FALSE;
  bLeakTest1Mode := FALSE;
  bLeakTest2Mode := TRUE;
  bBreakTestMode := FALSE;
  bJogMode := FALSE;
  bHandMode := FALSE;
ELSIF bBreakTestClicked THEN
  bBreakTestClicked := FALSE;
  bEnduranceRunMode := FALSE;
  bLeakTest1Mode := FALSE;
  bLeakTest2Mode := FALSE;
  bBreakTestMode := TRUE;
  bJogMode := FALSE;
  bHandMode := FALSE;
ELSIF bJogClicked THEN
  bJogClicked := FALSE;
  bEnduranceRunMode := FALSE;
  bLeakTest1Mode := FALSE;
  bLeakTest2Mode := FALSE;
  bBreakTestMode := FALSE;
  bJogMode := TRUE;
  bHandMode := FALSE;
ELSIF bHandClicked THEN
  bHandClicked := FALSE;
  bEnduranceRunMode := FALSE;
  bLeakTest1Mode := FALSE;
  bLeakTest2Mode := FALSE;
  bBreakTestMode := FALSE;
  bJogMode := FALSE;
  bHandMode := TRUE;
END_IF

IF bJogCounterCyl1_Clicked THEN
  bJogCounterCyl1_Clicked := FALSE;
  bJogCounterCyl1_Active := TRUE;
  bJogCounterCyl2_Active := FALSE;
  bJogCounterCyl3_Active := FALSE;
  bJogCounterCyl4_Active := FALSE;
ELSIF bJogCounterCyl2_Clicked THEN
  bJogCounterCyl2_Clicked := FALSE;
  bJogCounterCyl1_Active := FALSE;
  bJogCounterCyl2_Active := TRUE;
  bJogCounterCyl3_Active := FALSE;
  bJogCounterCyl4_Active := FALSE;
ELSIF bJogCounterCyl3_Clicked THEN
  bJogCounterCyl3_Clicked := FALSE;
  bJogCounterCyl1_Active := FALSE;
  bJogCounterCyl2_Active := FALSE;
  bJogCounterCyl3_Active := TRUE;
  bJogCounterCyl4_Active := FALSE;
ELSIF bJogCounterCyl4_Clicked THEN
  bJogCounterCyl4_Clicked := FALSE;
  bJogCounterCyl1_Active := FALSE;
  bJogCounterCyl2_Active := FALSE;
  bJogCounterCyl3_Active := FALSE;
  bJogCounterCyl4_Active := TRUE;
END_IF

METHOD FB_init : BOOL
VAR_INPUT
	bInitRetains : BOOL; // if TRUE, the retain variables are initialized (warm start / cold start)
	bInCopyCode : BOOL;  // if TRUE, the instance afterwards gets moved into the copy code (online change)
  
	itfOpMode:  I_OP_MODE_PAUSE;
END_VAR
THIS^.itfOpMode := itfOpMode;
END_METHOD

METHOD M_ResetModeSelection : BOOL
VAR_INPUT
END_VAR
M_ResetModeSelection := TRUE
                        AND NOT THIS^.bEnduranceRunMode
                        AND NOT THIS^.bLeakTest1Mode
                        AND NOT THIS^.bLeakTest2Mode
                        AND NOT THIS^.bBreakTestMode
                        AND NOT THIS^.bJogMode
                        AND NOT THIS^.bHandMode
                        AND NOT THIS^.bJogCounterCyl1_Active
                        AND NOT THIS^.bJogCounterCyl2_Active
                        AND NOT THIS^.bJogCounterCyl3_Active
                        AND NOT THIS^.bJogCounterCyl4_Active;

THIS^.bEnduranceRunMode := FALSE;
THIS^.bLeakTest1Mode := FALSE;
THIS^.bLeakTest2Mode := FALSE;
THIS^.bBreakTestMode := FALSE;
THIS^.bJogMode := FALSE;
THIS^.bHandMode := FALSE;
THIS^.bJogCounterCyl1_Active := FALSE;
THIS^.bJogCounterCyl2_Active := FALSE;
THIS^.bJogCounterCyl3_Active := FALSE;
THIS^.bJogCounterCyl4_Active := FALSE;
END_METHOD

{warning 'Methodenimplementierung hinzufügen'}
(*=== Method: M_Run  ============================================

 @brief: Here is the global code (Timer, Event, Flange,...)*)
METHOD M_Run
END_METHOD

PROPERTY P_BreakPressureDetSelected : BOOL
GET
P_BreakPressureDetSelected := THIS^.bBreakTestMode;
END_GET
END_PROPERTY

PROPERTY P_EnduranceRunSelected : BOOL
GET
P_EnduranceRunSelected := THIS^.bEnduranceRunMode;
END_GET
END_PROPERTY

{warning 'Eigenschaftenimplementierung hinzufügen'}
(*=== Property: P_Event  ============================================

 @param [set]: 	Set the Structure "ST_EVENT" from another Object
 @param [get]: 	Return the Structure "ST_EVENT", it contains the actual 
					event of the Object *)
PROPERTY P_Event : GenLib.ST_EVENT
GET
END_GET
SET
END_SET
END_PROPERTY

{warning 'Eigenschaftenimplementierung hinzufügen'}
(*=== Property: P_FullObjectPath  ============================================

 @param [set]: 	Set the Object Path (Clear String of Object)
 @param [get]: 	Return the Objectpath *)
PROPERTY P_FullObjectPath : STRING
GET
END_GET
SET
END_SET
END_PROPERTY

{warning 'Eigenschaftenimplementierung hinzufügen'}
(*=== Property: P_Global_Ack  ============================================

 @param [set]: 	Set the Bit for Ack from another Object
 @param [get]: 	Return the state of Ack Bit*)
PROPERTY P_Global_Ack : BOOL
GET
END_GET
SET
END_SET
END_PROPERTY

{warning 'Eigenschaftenimplementierung hinzufügen'}
(*=== Property: P_GlobalID  ============================================

 @param [set]: 	-
 @param [get]: 	Return the string of instance path*)
PROPERTY P_GlobalID : STRING
GET
END_GET
END_PROPERTY

PROPERTY P_HandSelected : BOOL
GET
P_HandSelected := THIS^.bHandMode;
END_GET
END_PROPERTY

{warning 'Eigenschaftenimplementierung hinzufügen'}
PROPERTY P_JogCounterCyl1_Active : BOOL
GET
P_JogCounterCyl1_Active := THIS^.bJogCounterCyl1_Active;
END_GET
END_PROPERTY

PROPERTY P_JogCounterCyl2_Active : BOOL
GET
P_JogCounterCyl2_Active := THIS^.bJogCounterCyl2_Active;
END_GET
END_PROPERTY

PROPERTY P_JogCounterCyl3_Active : BOOL
GET
P_JogCounterCyl3_Active := THIS^.bJogCounterCyl3_Active;
END_GET
END_PROPERTY

PROPERTY P_JogCounterCyl4_Active : BOOL
GET
P_JogCounterCyl4_Active := THIS^.bJogCounterCyl4_Active;
END_GET
END_PROPERTY

PROPERTY P_JogSelected : BOOL
GET
P_JogSelected := THIS^.bJogMode;
END_GET
END_PROPERTY

PROPERTY P_LeakTest1Selected : BOOL
GET
P_LeakTest1Selected := THIS^.bLeakTest1Mode;
END_GET
END_PROPERTY

PROPERTY P_LeakTest2Selected : BOOL
GET
P_LeakTest2Selected := THIS^.bLeakTest2Mode;
END_GET
END_PROPERTY

END_FUNCTION_BLOCK

// ---- MODULE/HMI/POU/FB_HMI_CTRL_ADS.TcPOU
FUNCTION_BLOCK FB_HMI_CTRL_ADS IMPLEMENTS I_HMI_CTRL
VAR_INPUT
  bLifeBit:                                               BOOL;
  bAdsConnected:                                          BOOL;
  bReady:                                                 BOOL;
  bBusy:                                                  BOOL;
END_VAR
VAR_OUTPUT
  liFreeSpaceOnC:                                         LINT;
END_VAR
VAR //General
	{attribute 'instance-path'} 
  {attribute 'noinit'} 
	strInstancePath:									                      STRING;
	bInit: 												                          BOOL:=TRUE;
	strFullObjectPath: 								                      STRING;
	stEvent:											                          ST_EVENT;
	bAck:												                            BOOL;
	
END_VAR
VAR   // From FB_init	
	itfOpMode:											                        I_OP_MODE; 
  itfEventLogger:                                         I_EVENT_LOGGER; 
END_VAR                                      				
VAR	// Step chain control                				
  eSeq, eLastSeq, eNextSeq:					                      E_SEQ_HMI; 
                  				
  //eActiveSeqState, eLastActiveSeqState:                 E_SEQ_GENERAL;
	(*
  iInternalSeqStateCase, iLastInternalSeqStateCase:       INT:=0;       
	tonDelay, tonTimeOut, tonStepTime:						          TON;
	tDelay:													                        TIME := T#100MS;
	tTimeOut:												                        TIME := T#100MS;
	tTimeOutExt:											                      TIME := T#100MS;
	bDelayActive, bTimeOutActiveQuit, bTimeOutActiveNoQuit:	BOOL;//Timer Option
	bActiveStep, bDebugAcitve, bDebugNext:					        BOOL;//Debug Option
	i:														                          INT;
 	iError:													                        INT; //ERROR-CODE                    	                   		
	listLastSteps:											                    ARRAY[0..49] OF ST_LAST_STEPS;	
	strExtraInfo:											                      STRING; 
	eStep_Type:												                      E_STEP_STATE_TYPE; 
	bDebugModeActive:										                    BOOL;   
	bWaitForBreakpoint:										                  BOOL;
	bBreakpointActive:										                  BOOL;
	bDebugResume:											                      BOOL;   
	listBreakpoint:											                    ARRAY[0..10] OF  INT;    
*)
i:														                            INT;
stSeqCtrlGeneral:											                    ST_SEQ_CTRL_GEN;     	
END_VAR                                             		
VAR                                                 		
	bMethodeFromExtStarted:									                BOOL;
	bMethodeFromExtActive:									                BOOL;
	bMethodeFromExtDone:									                  BOOL;
	strTemp:												                        STRING;
END_VAR   
VAR
  // From ADS
  bDBLifeBit:                                             BOOL;
  // To ADS
  bOpenKeyboard:                                          BOOL;
  bStartHMI:                                              BOOL;
  bCloseHMI:                                              BOOL;
  bShutdownPc:                                            BOOL;
  bRestartPc:                                             BOOL;
  udiFreeSpaceOnC:                                        UDINT;
END_VAR                  	
VAR_TEMP                    	
	iTemp:										                              INT;
END_VAR

// Set FBs and Interfaces ready after switch internal step
IF stSeqCtrlGeneral.iInternalSeqStateCase <> stSeqCtrlGeneral.iLastInternalSeqStateCase AND NOT stSeqCtrlGeneral.bExitSetReadyState THEN
  IF TRUE
  THEN
    stSeqCtrlGeneral.bExitSetReadyState := TRUE;
  ELSE
    RETURN;
  END_IF
END_IF

stSeqCtrlGeneral.strObject := F_CreateObjectName(strInstancePath);

udiFreeSpaceOnC := TO_UDINT(liFreeSpaceOnC);

// First method call
_m_SequenceManager();
//_m_SaveLastStep();

CASE eSeq OF 
  E_SEQ_HMI.BASE:;
  
	E_SEQ_HMI.INIT: _m_Seq_INIT();
		IF TRUE
		AND (stSeqCtrlGeneral.eActiveSeqState = E_SEQ_GENERAL.DONE) 
		THEN
			eSeq := E_SEQ_HMI.BASE;
		END_IF
		
	E_SEQ_HMI.SETUP:;
  
	// Process
  E_SEQ_HMI.START_HMI: _m_Seq_START_HMI();
    IF TRUE
		AND (stSeqCtrlGeneral.eActiveSeqState = E_SEQ_GENERAL.DONE) 
		THEN
			eSeq := E_SEQ_HMI.BASE;
		END_IF
    
  E_SEQ_HMI.CLOSE_HMI: _m_Seq_CLOSE_HMI();
    IF TRUE
		AND (stSeqCtrlGeneral.eActiveSeqState = E_SEQ_GENERAL.DONE) 
		THEN
			eSeq := E_SEQ_HMI.BASE;
		END_IF
    
  E_SEQ_HMI.PC_REBOOT: _m_Seq_PC_REBOOT();
    IF TRUE
		AND (stSeqCtrlGeneral.eActiveSeqState = E_SEQ_GENERAL.DONE) 
		THEN
			eSeq := E_SEQ_HMI.BASE;
		END_IF
    
  E_SEQ_HMI.PC_SHUTDOWN: _m_Seq_PC_SHUTDOWN();
    IF TRUE
		AND (stSeqCtrlGeneral.eActiveSeqState = E_SEQ_GENERAL.DONE) 
		THEN
			eSeq := E_SEQ_HMI.BASE;
		END_IF
    
  E_SEQ_HMI.SHOW_WIN_KEYBOARD: _m_Seq_SHOW_WIN_KEYBOARD();
    IF TRUE
		AND (stSeqCtrlGeneral.eActiveSeqState = E_SEQ_GENERAL.DONE) 
		THEN
			eSeq := E_SEQ_HMI.BASE;
		END_IF
    
  E_SEQ_HMI.HIDE_WIN_KEYBOARD: _m_Seq_HIDE_WIN_KEYBOARD();
    IF TRUE
		AND (stSeqCtrlGeneral.eActiveSeqState = E_SEQ_GENERAL.DONE) 
		THEN
			eSeq := E_SEQ_HMI.BASE;
		END_IF

  // End
	E_SEQ_HMI.END:;
	E_SEQ_HMI.ERROR_SEQ:;	
END_CASE

strTemp:=TO_STRING(eSeq);

METHOD PRIVATE _m_DebugManager
VAR_INPUT
	iStepID: int;
END_VAR
IF TRUE
AND THIS^.stSeqCtrlGeneral.bDebugModeActive 
AND NOT THIS^.stSeqCtrlGeneral.bActiveStep
THEN


THIS^.stSeqCtrlGeneral.bBreakpointActive:=FALSE;

FOR i:=0 TO 10 DO
	
	IF TRUE
	AND iStepID=THIS^.stSeqCtrlGeneral.listBreakpoint[i] 
	AND iStepID<>0
	THEN
		EXIT;
	END_IF
END_FOR
IF (i<=10) THEN
	THIS^.stSeqCtrlGeneral.bBreakpointActive:=TRUE;
END_IF

END_IF
END_METHOD

METHOD PRIVATE _m_Delay : BOOL
VAR_INPUT
	DelayTime:	TIME;
END_VAR
THIS^.stSeqCtrlGeneral.bDelayActive:=TRUE;
THIS^.stSeqCtrlGeneral.tDelay:=DelayTime;
_m_Delay:=FALSE;
IF THIS^.stSeqCtrlGeneral.tonDelay.Q THEN
	_m_Delay:=TRUE;
END_IF
END_METHOD

METHOD PRIVATE _m_GeneralStepSetting : BOOL
VAR_INPUT
	StepType:			    	E_STEP_STATE_TYPE;
	InfoTextID:					STRING(20);
	EnableDebug:	   			BOOL;	
	
END_VAR
IF THIS^.stSeqCtrlGeneral.bActiveStep THEN
	THIS^.stSeqCtrlGeneral.eStep_Type:=StepType;
	THIS^.stSeqCtrlGeneral.strExtraInfo:= GenLib.F_RET_TXTLIST_ENTRY(strPortNr:='851',strID:='',strTxtLstName:=InfoTextID);
END_IF
END_METHOD

METHOD PRIVATE _m_SaveLastStep : BOOL
VAR_INPUT
END_VAR
VAR
	i: dint;
END_VAR
IF NOT THIS^.stSeqCtrlGeneral.bActiveStep THEN
	
	FOR i:=49 TO 1 BY -1 DO
			stSeqCtrlGeneral.listLastSteps[i].strStepName:=stSeqCtrlGeneral.listLastSteps[i-1].strStepName;
			stSeqCtrlGeneral.listLastSteps[i].tStepTime:=stSeqCtrlGeneral.listLastSteps[i-1].tStepTime;
			stSeqCtrlGeneral.listLastSteps[i].tDelayTime:=stSeqCtrlGeneral.listLastSteps[i-1].tDelayTime;
	END_FOR
	stSeqCtrlGeneral.listLastSteps[0].strStepName:=TO_STRING(THIS^.eSeq);
	stSeqCtrlGeneral.listLastSteps[1].tStepTime:=THIS^.stSeqCtrlGeneral.tonStepTime.ET;
	stSeqCtrlGeneral.listLastSteps[1].tStepTime:=THIS^.stSeqCtrlGeneral.tonDelay.ET;
ELSE
	stSeqCtrlGeneral.listLastSteps[0].tStepTime:=THIS^.stSeqCtrlGeneral.tonStepTime.ET;
	stSeqCtrlGeneral.listLastSteps[0].tDelayTime:=THIS^.stSeqCtrlGeneral.tonDelay.ET;	
END_IF
END_METHOD

METHOD PRIVATE _m_Seq_CLOSE_HMI : E_SEQ_PROCESS
VAR_INPUT
END_VAR
VAR
	ActiveSeq: STRING;
END_VAR
//THIS^._m_GeneralStepSetting(StepType:=E_STEP_STATE_TYPE.INIT,
ActiveSeq := TO_STRING(THIS^.eSeq);

CASE THIS^.stSeqCtrlGeneral.eActiveSeqState OF
E_SEQ_GENERAL.READY:;
	
E_SEQ_GENERAL.EXECUTE:;
	IF TRUE
	THEN
		THIS^.stSeqCtrlGeneral.eActiveSeqState := E_SEQ_GENERAL.RESET;
	END_IF
  
E_SEQ_GENERAL.RESET:;
	THIS^.stSeqCtrlGeneral.iInternalSeqStateCase := 0;
	IF TRUE
	THEN
		THIS^.stSeqCtrlGeneral.eActiveSeqState := E_SEQ_GENERAL.BUSY;
	END_IF
  
E_SEQ_GENERAL.BUSY:;
	CASE THIS^.stSeqCtrlGeneral.iInternalSeqStateCase OF
    0:  // Execute
      IF TRUE 
      AND THIS^.bAdsConnected
      AND NOT THIS^.bBusy
      AND THIS^.bReady
			THEN 
        THIS^.bCloseHMI := TRUE;
        THIS^.stSeqCtrlGeneral.iInternalSeqStateCase := 10;
			END_IF

    10:	// Wait for done
      IF TRUE 
      AND NOT THIS^.bBusy
      AND THIS^.bReady
      AND NOT THIS^.bCloseHMI
			THEN 
        THIS^.stSeqCtrlGeneral.iInternalSeqStateCase := 1000;
			END_IF
      
    1000: // Exit step
      IF TRUE
      THEN
        THIS^.stSeqCtrlGeneral.iInternalSeqStateCase := 9999;
			END_IF
      
	ELSE
		THIS^.stSeqCtrlGeneral.eActiveSeqState := E_SEQ_GENERAL.DONE;  
	END_CASE
	THIS^.stSeqCtrlGeneral.strExtraInfo := CONCAT('Internal state: ', TO_STRING(THIS^.stSeqCtrlGeneral.iInternalSeqStateCase));

E_SEQ_GENERAL.DONE:;

E_SEQ_GENERAL.ERROR:;

E_SEQ_GENERAL.TIME_OUT:; 

ELSE
  THIS^.stSeqCtrlGeneral.eActiveSeqState := E_SEQ_GENERAL.ERROR;
END_CASE
END_METHOD

METHOD PRIVATE _m_Seq_HIDE_WIN_KEYBOARD : E_SEQ_PROCESS
VAR_INPUT
END_VAR
VAR
	ActiveSeq: STRING;
END_VAR
//THIS^._m_GeneralStepSetting(StepType:=E_STEP_STATE_TYPE.INIT,
ActiveSeq := TO_STRING(THIS^.eSeq);

CASE THIS^.stSeqCtrlGeneral.eActiveSeqState OF
E_SEQ_GENERAL.READY:;
	
E_SEQ_GENERAL.EXECUTE:;
	IF TRUE
	THEN
		THIS^.stSeqCtrlGeneral.eActiveSeqState := E_SEQ_GENERAL.RESET;
	END_IF
  
E_SEQ_GENERAL.RESET:;
	THIS^.stSeqCtrlGeneral.iInternalSeqStateCase := 0;
	IF TRUE
	THEN
		THIS^.stSeqCtrlGeneral.eActiveSeqState := E_SEQ_GENERAL.BUSY;
	END_IF
  
E_SEQ_GENERAL.BUSY:;
	CASE THIS^.stSeqCtrlGeneral.iInternalSeqStateCase OF
    0:  // Execute
      IF TRUE 
      AND THIS^.bAdsConnected
      AND NOT THIS^.bBusy
      AND THIS^.bReady
			THEN 
        THIS^.bOpenKeyboard := FALSE;
        THIS^.stSeqCtrlGeneral.iInternalSeqStateCase := 1000;
			END_IF
      
    1000: // Exit step
      IF TRUE
      THEN
        THIS^.stSeqCtrlGeneral.iInternalSeqStateCase := 9999;
			END_IF
      
	ELSE
		THIS^.stSeqCtrlGeneral.eActiveSeqState := E_SEQ_GENERAL.DONE;  
	END_CASE
	THIS^.stSeqCtrlGeneral.strExtraInfo := CONCAT('Internal state: ', TO_STRING(THIS^.stSeqCtrlGeneral.iInternalSeqStateCase));

E_SEQ_GENERAL.DONE:;

E_SEQ_GENERAL.ERROR:;

E_SEQ_GENERAL.TIME_OUT:; 

ELSE
  THIS^.stSeqCtrlGeneral.eActiveSeqState := E_SEQ_GENERAL.ERROR;
END_CASE
END_METHOD

METHOD PRIVATE _m_Seq_INIT : E_SEQ_PROCESS
VAR_INPUT
END_VAR
VAR
	ActiveSeq: STRING;
END_VAR
VAR
	
END_VAR
//THIS^._m_GeneralStepSetting(StepType:=E_STEP_STATE_TYPE.INIT,
ActiveSeq := TO_STRING(THIS^.eSeq);

CASE THIS^.stSeqCtrlGeneral.eActiveSeqState OF
E_SEQ_GENERAL.READY:;
	
E_SEQ_GENERAL.EXECUTE:;
	IF TRUE
	THEN
		THIS^.stSeqCtrlGeneral.eActiveSeqState := E_SEQ_GENERAL.RESET;
	END_IF
E_SEQ_GENERAL.RESET:;
	THIS^.stSeqCtrlGeneral.iInternalSeqStateCase := 0;
	IF TRUE
	THEN
		THIS^.stSeqCtrlGeneral.eActiveSeqState := E_SEQ_GENERAL.BUSY;
	END_IF
E_SEQ_GENERAL.BUSY:;
	CASE THIS^.stSeqCtrlGeneral.iInternalSeqStateCase OF
		0:	// Entrance step
      IF TRUE
			THEN 
        THIS^.bOpenKeyboard := FALSE;
        THIS^.bCloseHMI := FALSE;
        THIS^.bShutdownPc := FALSE;
        THIS^.bRestartPc := FALSE;
				THIS^.stSeqCtrlGeneral.iInternalSeqStateCase := 1000;
			END_IF
      
    1000:	// Exit step
      IF TRUE
			THEN
        THIS^.stSeqCtrlGeneral.iInternalSeqStateCase := 9999;
      END_IF
      
	ELSE
		THIS^.stSeqCtrlGeneral.eActiveSeqState := E_SEQ_GENERAL.DONE;  
	END_CASE
	THIS^.stSeqCtrlGeneral.strExtraInfo := CONCAT('Internal state: ', TO_STRING(THIS^.stSeqCtrlGeneral.iInternalSeqStateCase));
E_SEQ_GENERAL.DONE:;
E_SEQ_GENERAL.ERROR:;
E_SEQ_GENERAL.TIME_OUT:; 

IF TRUE
AND THIS^.stSeqCtrlGeneral.bTimeOutActiveQuit 
THEN
  THIS^.stSeqCtrlGeneral.strExtraInfo := 'Bitte quittieren und erneut testen';
  IF TRUE
  //AND itfOpMode.P_QUIT
  THEN
    THIS^.stSeqCtrlGeneral.eActiveSeqState := E_SEQ_GENERAL.EXECUTE;
	END_IF
  
END_IF

ELSE
  THIS^.stSeqCtrlGeneral.eActiveSeqState := E_SEQ_GENERAL.ERROR;
END_CASE
END_METHOD

METHOD PRIVATE _m_Seq_PC_REBOOT : E_SEQ_PROCESS
VAR_INPUT
END_VAR
VAR
	ActiveSeq: STRING;
END_VAR
//THIS^._m_GeneralStepSetting(StepType:=E_STEP_STATE_TYPE.INIT,
ActiveSeq := TO_STRING(THIS^.eSeq);

CASE THIS^.stSeqCtrlGeneral.eActiveSeqState OF
E_SEQ_GENERAL.READY:;
	
E_SEQ_GENERAL.EXECUTE:;
	IF TRUE
	THEN
		THIS^.stSeqCtrlGeneral.eActiveSeqState := E_SEQ_GENERAL.RESET;
	END_IF
  
E_SEQ_GENERAL.RESET:;
	THIS^.stSeqCtrlGeneral.iInternalSeqStateCase := 0;
	IF TRUE
	THEN
		THIS^.stSeqCtrlGeneral.eActiveSeqState := E_SEQ_GENERAL.BUSY;
	END_IF
  
E_SEQ_GENERAL.BUSY:;
	CASE THIS^.stSeqCtrlGeneral.iInternalSeqStateCase OF
    0:  // Execute
      IF TRUE 
      AND THIS^.bAdsConnected
      AND NOT THIS^.bBusy
      AND THIS^.bReady
			THEN 
        THIS^.bRestartPc := TRUE;
        THIS^.stSeqCtrlGeneral.iInternalSeqStateCase := 10;
			END_IF

    10:	// Wait for done
      IF TRUE 
      AND NOT THIS^.bBusy
      AND THIS^.bReady
      AND NOT THIS^.bRestartPc
			THEN 
        THIS^.stSeqCtrlGeneral.iInternalSeqStateCase := 1000;
			END_IF
      
    1000: // Exit step
      IF TRUE
      THEN
        THIS^.stSeqCtrlGeneral.iInternalSeqStateCase := 9999;
			END_IF
      
	ELSE
		THIS^.stSeqCtrlGeneral.eActiveSeqState := E_SEQ_GENERAL.DONE;  
	END_CASE
	THIS^.stSeqCtrlGeneral.strExtraInfo := CONCAT('Internal state: ', TO_STRING(THIS^.stSeqCtrlGeneral.iInternalSeqStateCase));

E_SEQ_GENERAL.DONE:;

E_SEQ_GENERAL.ERROR:;

E_SEQ_GENERAL.TIME_OUT:; 

ELSE
  THIS^.stSeqCtrlGeneral.eActiveSeqState := E_SEQ_GENERAL.ERROR;
END_CASE
END_METHOD

METHOD PRIVATE _m_Seq_PC_SHUTDOWN : E_SEQ_PROCESS
VAR_INPUT
END_VAR
VAR
	ActiveSeq: STRING;
END_VAR
//THIS^._m_GeneralStepSetting(StepType:=E_STEP_STATE_TYPE.INIT,
ActiveSeq := TO_STRING(THIS^.eSeq);

CASE THIS^.stSeqCtrlGeneral.eActiveSeqState OF
E_SEQ_GENERAL.READY:;
	
E_SEQ_GENERAL.EXECUTE:;
	IF TRUE
	THEN
		THIS^.stSeqCtrlGeneral.eActiveSeqState := E_SEQ_GENERAL.RESET;
	END_IF
  
E_SEQ_GENERAL.RESET:;
	THIS^.stSeqCtrlGeneral.iInternalSeqStateCase := 0;
	IF TRUE
	THEN
		THIS^.stSeqCtrlGeneral.eActiveSeqState := E_SEQ_GENERAL.BUSY;
	END_IF
  
E_SEQ_GENERAL.BUSY:;
	CASE THIS^.stSeqCtrlGeneral.iInternalSeqStateCase OF
    0:  // Execute
      IF TRUE 
      AND THIS^.bAdsConnected
      AND NOT THIS^.bBusy
      AND THIS^.bReady
			THEN 
        THIS^.bShutdownPc := TRUE;
        THIS^.stSeqCtrlGeneral.iInternalSeqStateCase := 10;
			END_IF

    10:	// Wait for done
      IF TRUE 
      AND NOT THIS^.bBusy
      AND THIS^.bReady
      AND NOT THIS^.bShutdownPc
			THEN 
        THIS^.stSeqCtrlGeneral.iInternalSeqStateCase := 1000;
			END_IF
      
    1000: // Exit step
      IF TRUE
      THEN
        THIS^.stSeqCtrlGeneral.iInternalSeqStateCase := 9999;
			END_IF
      
	ELSE
		THIS^.stSeqCtrlGeneral.eActiveSeqState := E_SEQ_GENERAL.DONE;  
	END_CASE
	THIS^.stSeqCtrlGeneral.strExtraInfo := CONCAT('Internal state: ', TO_STRING(THIS^.stSeqCtrlGeneral.iInternalSeqStateCase));

E_SEQ_GENERAL.DONE:;

E_SEQ_GENERAL.ERROR:;

E_SEQ_GENERAL.TIME_OUT:; 

ELSE
  THIS^.stSeqCtrlGeneral.eActiveSeqState := E_SEQ_GENERAL.ERROR;
END_CASE
END_METHOD

METHOD PRIVATE _m_Seq_SHOW_WIN_KEYBOARD : E_SEQ_PROCESS
VAR_INPUT
END_VAR
VAR
	ActiveSeq: STRING;
END_VAR
//THIS^._m_GeneralStepSetting(StepType:=E_STEP_STATE_TYPE.INIT,
ActiveSeq := TO_STRING(THIS^.eSeq);

CASE THIS^.stSeqCtrlGeneral.eActiveSeqState OF
E_SEQ_GENERAL.READY:;
	
E_SEQ_GENERAL.EXECUTE:;
	IF TRUE
	THEN
		THIS^.stSeqCtrlGeneral.eActiveSeqState := E_SEQ_GENERAL.RESET;
	END_IF
  
E_SEQ_GENERAL.RESET:;
	THIS^.stSeqCtrlGeneral.iInternalSeqStateCase := 0;
	IF TRUE
	THEN
		THIS^.stSeqCtrlGeneral.eActiveSeqState := E_SEQ_GENERAL.BUSY;
	END_IF
  
E_SEQ_GENERAL.BUSY:;
	CASE THIS^.stSeqCtrlGeneral.iInternalSeqStateCase OF
    0:  // Execute
      IF TRUE 
      AND THIS^.bAdsConnected
      AND NOT THIS^.bBusy
      AND THIS^.bReady
			THEN 
        THIS^.bOpenKeyboard := TRUE;
        THIS^.stSeqCtrlGeneral.iInternalSeqStateCase := 1000;
			END_IF
      
    1000: // Exit step
      IF TRUE
      THEN
        THIS^.stSeqCtrlGeneral.iInternalSeqStateCase := 9999;
			END_IF
      
	ELSE
		THIS^.stSeqCtrlGeneral.eActiveSeqState := E_SEQ_GENERAL.DONE;  
	END_CASE
	THIS^.stSeqCtrlGeneral.strExtraInfo := CONCAT('Internal state: ', TO_STRING(THIS^.stSeqCtrlGeneral.iInternalSeqStateCase));

E_SEQ_GENERAL.DONE:;

E_SEQ_GENERAL.ERROR:;

E_SEQ_GENERAL.TIME_OUT:; 

ELSE
  THIS^.stSeqCtrlGeneral.eActiveSeqState := E_SEQ_GENERAL.ERROR;
END_CASE
END_METHOD

METHOD PRIVATE _m_Seq_START_HMI : E_SEQ_PROCESS
VAR_INPUT
END_VAR
VAR
	ActiveSeq: STRING;
END_VAR
//THIS^._m_GeneralStepSetting(StepType:=E_STEP_STATE_TYPE.INIT,
ActiveSeq := TO_STRING(THIS^.eSeq);

CASE THIS^.stSeqCtrlGeneral.eActiveSeqState OF
E_SEQ_GENERAL.READY:;
	
E_SEQ_GENERAL.EXECUTE:;
	IF TRUE
	THEN
		THIS^.stSeqCtrlGeneral.eActiveSeqState := E_SEQ_GENERAL.RESET;
	END_IF
  
E_SEQ_GENERAL.RESET:;
	THIS^.stSeqCtrlGeneral.iInternalSeqStateCase := 0;
	IF TRUE
	THEN
		THIS^.stSeqCtrlGeneral.eActiveSeqState := E_SEQ_GENERAL.BUSY;
	END_IF
  
E_SEQ_GENERAL.BUSY:;
	CASE THIS^.stSeqCtrlGeneral.iInternalSeqStateCase OF
    0:  // Execute
      IF TRUE 
      AND THIS^.bAdsConnected
      AND NOT THIS^.bBusy
      AND THIS^.bReady
			THEN 
        THIS^.bStartHMI := TRUE;
        THIS^.stSeqCtrlGeneral.iInternalSeqStateCase := 10;
			END_IF

    10:	// Wait for done
      IF TRUE 
      AND NOT THIS^.bBusy
      AND THIS^.bReady
      AND NOT THIS^.bStartHMI
			THEN 
        THIS^.stSeqCtrlGeneral.iInternalSeqStateCase := 1000;
			END_IF
      
    1000: // Exit step
      IF TRUE
      THEN
        THIS^.stSeqCtrlGeneral.iInternalSeqStateCase := 9999;
			END_IF
      
	ELSE
		THIS^.stSeqCtrlGeneral.eActiveSeqState := E_SEQ_GENERAL.DONE;  
	END_CASE
	THIS^.stSeqCtrlGeneral.strExtraInfo := CONCAT('Internal state: ', TO_STRING(THIS^.stSeqCtrlGeneral.iInternalSeqStateCase));

E_SEQ_GENERAL.DONE:;

E_SEQ_GENERAL.ERROR:;

E_SEQ_GENERAL.TIME_OUT:; 

ELSE
  THIS^.stSeqCtrlGeneral.eActiveSeqState := E_SEQ_GENERAL.ERROR;
END_CASE
END_METHOD

METHOD PRIVATE _m_SequenceManager
VAR_INPUT
END_VAR
IF FALSE
//AND THIS^.eActiveSeqState=DONE 
AND eLastSeq<>eSeq
THEN
	IF THIS^.stSeqCtrlGeneral.eActiveSeqState<>E_SEQ_GENERAL.EXECUTE THEN
		THIS^.stSeqCtrlGeneral.eActiveSeqState:=E_SEQ_GENERAL.READY;
	END_IF
END_IF

eSeq := eNextSeq;

//DelayTimer und TimeOut Timer verwalten
stSeqCtrlGeneral.bActiveStep:=	TRUE
				AND eLastSeq					=	eSeq
				AND stSeqCtrlGeneral.eLastActiveSeqState			=	stSeqCtrlGeneral.eActiveSeqState
				AND	stSeqCtrlGeneral.iLastInternalSeqStateCase	=	stSeqCtrlGeneral.iInternalSeqStateCase
				;
			
IF NOT stSeqCtrlGeneral.bActiveStep THEN
	stSeqCtrlGeneral.bDelayActive:=FALSE;
	stSeqCtrlGeneral.bTimeOutActiveQuit:=FALSE;
	stSeqCtrlGeneral.bTimeOutActiveNoQuit:=FALSE;
  THIS^.stSeqCtrlGeneral.strExtraInfo:='';
END_IF

_m_SaveLastStep();
stSeqCtrlGeneral.tonDelay	(IN:=stSeqCtrlGeneral.bActiveStep AND stSeqCtrlGeneral.bDelayActive, 		PT:=stSeqCtrlGeneral.tDelay);
stSeqCtrlGeneral.tonTimeOut	(IN:=stSeqCtrlGeneral.bActiveStep AND (stSeqCtrlGeneral.bTimeOutActiveNoQuit OR stSeqCtrlGeneral.bTimeOutActiveQuit), 	PT:=stSeqCtrlGeneral.tTimeOut);
stSeqCtrlGeneral.tonStepTime	(IN:= stSeqCtrlGeneral.bActiveStep, PT:= T#24H);

IF stSeqCtrlGeneral.tonTimeOut.Q  THEN
	stSeqCtrlGeneral.eActiveSeqState:=E_SEQ_GENERAL.TIME_OUT;
END_IF

IF stSeqCtrlGeneral.iError<>0 THEN
	eSeq:=E_SEQ_HMI.ERROR_SEQ;
END_IF



eLastSeq					:=	eSeq;
stSeqCtrlGeneral.eLastActiveSeqState			:=	stSeqCtrlGeneral.eActiveSeqState;
stSeqCtrlGeneral.iLastInternalSeqStateCase	:=	stSeqCtrlGeneral.iInternalSeqStateCase;

// Reset set ready state
IF THIS^.stSeqCtrlGeneral.bExitSetReadyState THEN
  THIS^.stSeqCtrlGeneral.bExitSetReadyState := FALSE;
END_IF
END_METHOD

METHOD PRIVATE _m_TimeOut : BOOL
VAR_INPUT
	bTimeoutActiveToQuit:	BOOL;
	bTimeOutActiveNoQuit:	BOOL;
	tTimeOut:				TIME;	
END_VAR
THIS^.stSeqCtrlGeneral.bTimeOutActiveQuit:=	bTimeoutActiveToQuit;
THIS^.stSeqCtrlGeneral.bTimeOutActiveNoQuit:=	bTimeOutActiveNoQuit;
THIS^.stSeqCtrlGeneral.tTimeOut:=			tTimeOut;
_m_TimeOut:=FALSE;
IF THIS^.stSeqCtrlGeneral.tonTimeOut.Q THEN
	_m_TimeOut:=TRUE;
END_IF
END_METHOD

METHOD FB_init : BOOL
VAR_INPUT
	bInitRetains : BOOL; // if TRUE, the retain variables are initialized (warm start / cold start)
	bInCopyCode : BOOL;  // if TRUE, the instance afterwards gets moved into the copy code (online change)
  
  itfOpMode:											                        I_OP_MODE; 
  itfEventLogger:                                         I_EVENT_LOGGER; 
END_VAR
THIS^.itfOpMode := itfOpMode;
THIS^.itfEventLogger := itfEventLogger;
END_METHOD

METHOD M_CloseHMI : BOOL
M_CloseHMI := THIS^.stSeqCtrlGeneral.eActiveSeqState = E_SEQ_GENERAL.DONE
              AND NOT THIS^.bCloseHMI;
              
// General
IF THIS^.stSeqCtrlGeneral.eActiveSeqState = E_SEQ_GENERAL.READY THEN
  THIS^.eNextSeq := E_SEQ_HMI.CLOSE_HMI;
  THIS^.stSeqCtrlGeneral.eActiveSeqState := E_SEQ_GENERAL.EXECUTE;
END_IF
END_METHOD

METHOD M_HideWinKeyboard : BOOL
M_HideWinKeyboard := THIS^.stSeqCtrlGeneral.eActiveSeqState = E_SEQ_GENERAL.DONE
                     AND NOT THIS^.bOpenKeyboard;

// General
IF THIS^.stSeqCtrlGeneral.eActiveSeqState = E_SEQ_GENERAL.READY THEN
  THIS^.eNextSeq := E_SEQ_HMI.HIDE_WIN_KEYBOARD;
  THIS^.stSeqCtrlGeneral.eActiveSeqState := E_SEQ_GENERAL.EXECUTE;
END_IF
END_METHOD

METHOD M_PCReboot : BOOL
M_PCReboot := THIS^.stSeqCtrlGeneral.eActiveSeqState = E_SEQ_GENERAL.DONE
              AND NOT THIS^.bRestartPc;

// General
IF THIS^.stSeqCtrlGeneral.eActiveSeqState = E_SEQ_GENERAL.READY THEN
  THIS^.eNextSeq := E_SEQ_HMI.PC_REBOOT;
  THIS^.stSeqCtrlGeneral.eActiveSeqState := E_SEQ_GENERAL.EXECUTE;
END_IF
END_METHOD

METHOD M_PCShutdown : BOOL
M_PCShutdown := THIS^.stSeqCtrlGeneral.eActiveSeqState = E_SEQ_GENERAL.DONE
                AND NOT THIS^.bShutdownPc;

// General
IF THIS^.stSeqCtrlGeneral.eActiveSeqState = E_SEQ_GENERAL.READY THEN
  THIS^.eNextSeq := E_SEQ_HMI.PC_SHUTDOWN;
  THIS^.stSeqCtrlGeneral.eActiveSeqState := E_SEQ_GENERAL.EXECUTE;
END_IF
END_METHOD

METHOD M_Reset : BOOL
VAR_INPUT
END_VAR
M_Reset := THIS^.stSeqCtrlGeneral.eActiveSeqState = E_SEQ_GENERAL.DONE;

// General
IF THIS^.stSeqCtrlGeneral.eActiveSeqState = E_SEQ_GENERAL.READY THEN
  THIS^.eNextSeq := E_SEQ_HMI.INIT;
  THIS^.stSeqCtrlGeneral.eActiveSeqState := E_SEQ_GENERAL.EXECUTE;
END_IF
END_METHOD

{warning 'Methodenimplementierung hinzufügen'}
(*=== Method: M_Run  ============================================

 @brief: Here is the global code (Timer, Event, Flange,...)*)
METHOD M_Run
END_METHOD

METHOD M_SetReady : BOOL
M_SetReady := TRUE
              AND THIS^.stSeqCtrlGeneral.eActiveSeqState = E_SEQ_GENERAL.READY
              AND THIS^.eSeq = E_SEQ_HMI.BASE;

THIS^.stSeqCtrlGeneral.eActiveSeqState := E_SEQ_GENERAL.READY;
THIS^.eNextSeq := E_SEQ_HMI.BASE;
END_METHOD

METHOD M_ShowWinKeyboard : BOOL
M_ShowWinKeyboard := THIS^.stSeqCtrlGeneral.eActiveSeqState = E_SEQ_GENERAL.DONE
                     AND THIS^.bOpenKeyboard;

// General
IF THIS^.stSeqCtrlGeneral.eActiveSeqState = E_SEQ_GENERAL.READY THEN
  THIS^.eNextSeq := E_SEQ_HMI.SHOW_WIN_KEYBOARD;
  THIS^.stSeqCtrlGeneral.eActiveSeqState := E_SEQ_GENERAL.EXECUTE;
END_IF
END_METHOD

METHOD M_StartHMI : BOOL
M_StartHMI := THIS^.stSeqCtrlGeneral.eActiveSeqState = E_SEQ_GENERAL.DONE
              AND NOT THIS^.bStartHMI;

// General
IF THIS^.stSeqCtrlGeneral.eActiveSeqState = E_SEQ_GENERAL.READY THEN
  THIS^.eNextSeq := E_SEQ_HMI.START_HMI;
  THIS^.stSeqCtrlGeneral.eActiveSeqState := E_SEQ_GENERAL.EXECUTE;
END_IF
END_METHOD

{warning 'Eigenschaftenimplementierung hinzufügen'}
PROPERTY P_ErrorMsg : STRING
GET
END_GET
SET
END_SET
END_PROPERTY

{warning 'Eigenschaftenimplementierung hinzufügen'}
(*=== Property: P_Event  ============================================

 @param [set]: 	Set the Structure "ST_EVENT" from another Object
 @param [get]: 	Return the Structure "ST_EVENT", it contains the actual 
					event of the Object *)
PROPERTY P_Event : GenLib.ST_EVENT
GET
END_GET
SET
END_SET
END_PROPERTY

{warning 'Eigenschaftenimplementierung hinzufügen'}
(*=== Property: P_FullObjectPath  ============================================

 @param [set]: 	Set the Object Path (Clear String of Object)
 @param [get]: 	Return the Objectpath *)
PROPERTY P_FullObjectPath : STRING
GET
END_GET
SET
END_SET
END_PROPERTY

{warning 'Eigenschaftenimplementierung hinzufügen'}
(*=== Property: P_Global_Ack  ============================================

 @param [set]: 	Set the Bit for Ack from another Object
 @param [get]: 	Return the state of Ack Bit*)
PROPERTY P_Global_Ack : BOOL
GET
END_GET
SET
END_SET
END_PROPERTY

{warning 'Eigenschaftenimplementierung hinzufügen'}
(*=== Property: P_GlobalID  ============================================

 @param [set]: 	-
 @param [get]: 	Return the string of instance path*)
PROPERTY P_GlobalID : STRING
GET
END_GET
END_PROPERTY

END_FUNCTION_BLOCK

// ---- MODULE/ACTOR_VALVE/HYDRAULIC_ACTOR/POU/FB_CYLINDER_DA_TESTDEV1.TcPOU
FUNCTION_BLOCK FB_CYLINDER_DA_TESTDEV1 IMPLEMENTS I_CYLINDER_DA_TESTDEV1
VAR_INPUT
  bDoableActing:                                          BOOL;
  lrCurrentPosAbs:                                        LREAL;
  rCurrentPressureInBar:                                  REAL;
  rCurrentPressureInBarA:                                 REAL;
  rCurrentPressureInBarB:                                 REAL;
  rCurrentLowPressureInBar:                               REAL;
  rCurrentLowPressureInBarA:                              REAL;
  rCurrentLowPressureInBarB:                              REAL;
  rCurrentReservoirPressureInBar:                         REAL;
  /// Cylinder piston surface A
  lrPistonSurfaceA:                                       LREAL;
  /// Cylinder piston surface B
  lrPistonSurfaceB:                                       LREAL;
  // Speed and Pressure regulation
  rSpeedRegulationFactor:                                 REAL;
  rSpeedRegulationTolerance:                              REAL;
  rPressureRegulationFactor:                              REAL;
  rPressureRegulationTolerance:                           REAL;
END_VAR
VAR //General
	{attribute 'instance-path'} 
  {attribute 'noinit'} 
	strInstancePath:									                      STRING;
	bInit: 												                          BOOL:=TRUE;
	strFullObjectPath: 								                      STRING;
	stEvent:											                          ST_EVENT;
	bAck:												                            BOOL;
	
END_VAR
VAR   // From FB_init	
	itfOpMode:											                        I_OP_MODE; 
  itfEventLogger:                                         I_EVENT_LOGGER;
  itfOpModeVisu:											                    I_OP_MODE_PAUSE_VISU;
  itfValve_CylCtrl:                                       I_VALVE_X_3_PROP;
  itfValve_LockA:                                         I_VALVE_X_2;
  itfValve_LockB:                                         I_VALVE_X_2;
  itfValve_AddPump2:                                      I_VALVE_X_2;
  itfValve_AddPump3:                                      I_VALVE_X_2;
  itfValve_AddPump4:                                      I_VALVE_X_2;
  itfValve_PressureReservoirAAdd:                         I_VALVE_X_2;
  itfValve_PressureReservoirBAdd:                         I_VALVE_X_2;
  itfValve_SensorBreakPressureAAdd:                       I_VALVE_X_2;
  itfValve_SensorBreakPressureBAdd:                       I_VALVE_X_2;
  itfShutOffValve_LowPressure:                            I_ENGINE_VALVE;
  itfValve_PressureLimit:                                 I_PRV_PROP;
  itfValve_LowPressureLimit:                              I_PRV_PROP;
  itfPumpMain:                                            I_PUMP;
  itfPump2:                                               I_PUMP;
  itfPump3:                                               I_PUMP;
  itfPump4:                                               I_PUMP;
  rEndPosTol:                                             REAL;
  /// Volume flow in l/min or dm³/min
  rPumpVolumeFlow:                                        REAL; // Volumenstrom
  /// Pump efficiency factor (0,5-1)
  rPumpEfficiencyFactor:                                  REAL; // Wirkungsgrad
END_VAR                                      				
VAR	// Step chain control                				
  eSeq, eLastSeq, eNextSeq:					                      E_SEQ_CYLINDER; 
                  				
  //eActiveSeqState, eLastActiveSeqState:                 E_SEQ_GENERAL;
	(*
  iInternalSeqStateCase, iLastInternalSeqStateCase:       INT:=0;       
	tonDelay, tonTimeOut, tonStepTime:						          TON;
	tDelay:													                        TIME := T#100MS;
	tTimeOut:												                        TIME := T#100MS;
	tTimeOutExt:											                      TIME := T#100MS;
	bDelayActive, bTimeOutActiveQuit, bTimeOutActiveNoQuit:	BOOL;//Timer Option
	bActiveStep, bDebugAcitve, bDebugNext:					        BOOL;//Debug Option
	i:														                          INT;
 	iError:													                        INT; //ERROR-CODE                    	                   		
	listLastSteps:											                    ARRAY[0..49] OF ST_LAST_STEPS;	
	strExtraInfo:											                      STRING; 
	eStep_Type:												                      E_STEP_STATE_TYPE; 
	bDebugModeActive:										                    BOOL;   
	bWaitForBreakpoint:										                  BOOL;
	bBreakpointActive:										                  BOOL;
	bDebugResume:											                      BOOL;   
	listBreakpoint:											                    ARRAY[0..10] OF  INT;    
*)
i:														                            INT;
ii:														                            INT;
iii:														                          INT;
stSeqCtrlGeneral:											                    ST_SEQ_CTRL_GEN;     	
END_VAR                                             		
VAR                                                 		
	bMethodeFromExtStarted:									                BOOL;
	bMethodeFromExtActive:									                BOOL;
	bMethodeFromExtDone:									                  BOOL;
	strTemp:												                        STRING;
END_VAR   
VAR
  stHMI:                                                  ST_HMI_CYLINDER;
  lrToSetPos:                                             LREAL;
  rTargetPressureInBarA:                                  REAL;
  rTargetPressureInBarB:                                  REAL;
  rTargetPressureInForceA:                                REAL;
  rTargetPressureInForceB:                                REAL;
  rTargetPressureInPercentA:                              REAL;
  rTargetPressureInPercentB:                              REAL;
  iTargetPressureAsValueA:                                INT;
  iTargetPressureAsValueB:                                INT;
  rSpeedInPercentToSet:                                   REAL;
  rSpeedInMmPerSToSet:                                    REAL;
  iSpeedAsValueToSet:                                     INT;
  rCurrentSpeedInMmPerS:                                  REAL;
  bStrokeLengthInitialized:                               BOOL;
  rStrokeLength:                                          REAL;
  lrPos:                                                  LREAL;
  lrPosZero:                                              LREAL;
  lrPosMax:                                               LREAL;
  bOpenReservoirA:                                        BOOL;
  bOpenReservoirB:                                        BOOL;
  bOpenChA:                                               BOOL;
	bOpenChB:                                               BOOL;
  bPump2Add:                                              BOOL;
  bPump3Add:                                              BOOL;
  bPump4Add:                                              BOOL;
  // Low Pressure
  bLowPressureEnabled:                                    BOOL;
  rLPTargetPressureInBarA:                                REAL;
  rLPTargetPressureInBarB:                                REAL;
  rLPTargetPressureInForceA:                              REAL;
  rLPTargetPressureInForceB:                              REAL;
  rLPTargetPressureInPercentA:                            REAL;
  rLPTargetPressureInPercentB:                            REAL;
  iLPTargetPressureAsValueA:                              INT;
  iLPTargetPressureAsValueB:                              INT;
END_VAR
VAR // Recording
  stRecord:											                          ST_RECORD;	 
	tonSaveInterval:											                  TON; 
	iCntRecord:											                        INT;	
	listGainRampData:									                      ARRAY[0..499] OF stMesswerte;
	stCurrentRamp:										                      stRampAnalytic;
	iCycleCntNormal:									                      INT;	
	uiLinRegStart:										                      UINT:=0;
  uiLinRegEnd:										                        UINT:=299; 
  rGainLimit_EndPos:                                      REAL:=0.1;
  lrLastPos:                                              LREAL;
  bJogCtrlBusy:                                           BOOL;
  bStartHPTrigger:                                        BOOL;
  bStartWPTrigger:                                        BOOL;
  bStopTrigger:                                           BOOL;
  bStartCalibrationClicked:                               BOOL;
  bStartLPCalibrationClicked:                             BOOL;
  // Speed
  listPosTable:                                           ARRAY[1..100] OF REAL;
  lrTotalPath:                                            LREAL;
  x:                                                      INT;
  xx:                                                     INT;
  iCorrectedSpeedValue:                                   INT;
  rCorrectedSpeedPercent:                                 REAL;
  bRegulation:                                            BOOL;
  bRegulationTrigger:                                     BOOL;
  uiRegulationSeq:                                        UINT := 0;
  bCorrectionTrigger:                                     BOOL;
  bRegulationBusy:                                        BOOL;
  uiPumpMultiplicator:                                    UINT;
  rCurrentForceInKN:                                      REAL;
  rCurrentForceInN:                                       REAL;
  rCurrentLowPressureForceInKN:                           REAL;
  rCurrentLowPressureForceInN:                            REAL;
  rActiveForce:                                           REAL;
  iCorrectedPressureAsValue:                              INT;
  bPressureRegulationTrigger:                             BOOL;
  bPressureRegulationBusy:                                BOOL;
  bPressureCorrectionTrigger:                             BOOL;
  uiPressureRegulationSeq:                                UINT := 0;
  bPressureRegulation:                                    BOOL;
END_VAR                   	
VAR_TEMP                    	
	iTemp:										INT;
END_VAR
VAR PERSISTENT
	listCylCalibration:                                     ARRAY[1..2, 1..100] OF LREAL;
  listCalibrationTable:                                   ARRAY[1..7] OF ST_CYL_CALIBRATION;
  listLPCylCalibration:                                   ARRAY[1..2, 1..100] OF LREAL;
  listLPCalibrationTable:                                 ARRAY[1..7] OF ST_CYL_CALIBRATION;
END_VAR

// Set FBs and Interfaces ready after switch internal step
IF stSeqCtrlGeneral.iInternalSeqStateCase <> stSeqCtrlGeneral.iLastInternalSeqStateCase AND NOT stSeqCtrlGeneral.bExitSetReadyState THEN
  IF TRUE
  AND itfValve_CylCtrl.M_SetReady()
  AND itfValve_LockA.M_SetReady()
  AND itfValve_LockB.M_SetReady()
  AND itfValve_AddPump2.M_SetReady()
  AND itfValve_AddPump3.M_SetReady()
  AND itfValve_AddPump4.M_SetReady()
  AND itfValve_PressureReservoirAAdd.M_SetReady()
  AND itfValve_PressureReservoirBAdd.M_SetReady()
  AND itfValve_SensorBreakPressureAAdd.M_SetReady()
  AND itfValve_SensorBreakPressureBAdd.M_SetReady()
  AND itfShutOffValve_LowPressure.M_SetReady()
  AND itfValve_PressureLimit.M_SetReady()
  AND itfValve_LowPressureLimit.M_SetReady()
  THEN
    stSeqCtrlGeneral.bExitSetReadyState := TRUE;
  ELSE
    RETURN;
  END_IF
END_IF

// Pump multiplicator
uiPumpMultiplicator := BOOL_TO_UINT(itfPumpMain.P_State)
                       + BOOL_TO_UINT(itfPump2.P_State AND itfValve_AddPump2.P_InWP1)
                       + BOOL_TO_UINT(itfPump3.P_State AND itfValve_AddPump3.P_InWP1)
                       + BOOL_TO_UINT(itfPump4.P_State AND itfValve_AddPump4.P_InWP1);
rCurrentForceInKN := P_CurrentForceInKN;
rCurrentForceInN := P_CurrentForceInKN * 1000;
rCurrentLowPressureForceInKN := P_CurrentLowPressureForceInN / 1000;
rCurrentLowPressureForceInN := P_CurrentLowPressureForceInN;
                       
                       
stSeqCtrlGeneral.strObjectPath := strInstancePath;
stSeqCtrlGeneral.strObject := F_CreateObjectName(strInstancePath);

// First method call
_m_SequenceManager();
//_m_SaveLastStep();
_m_SpeedRegulation();
_m_PressureRegulation();
_m_Recording();
_m_ManualOperation();
_m_PressureCalibration();
_m_HMI();

CASE eSeq OF 
  E_SEQ_CYLINDER.BASE:;
  
	E_SEQ_CYLINDER.INIT: _m_Seq_INIT();
		IF TRUE
		AND (stSeqCtrlGeneral.eActiveSeqState = E_SEQ_GENERAL.DONE) 
		THEN
			eSeq := E_SEQ_CYLINDER.BASE;
		END_IF
		
	E_SEQ_CYLINDER.SETUP:;
  
	// Process
  E_SEQ_CYLINDER.SET_MAX_POS: _m_Seq_SET_MAX_POS();
    IF TRUE
		AND (stSeqCtrlGeneral.eActiveSeqState = E_SEQ_GENERAL.DONE) 
		THEN
			eSeq := E_SEQ_CYLINDER.BASE;
		END_IF
  
  E_SEQ_CYLINDER.SET_WORK_PRESSURE: _m_Seq_SET_WORK_PRESSURE();
    IF TRUE
		AND (stSeqCtrlGeneral.eActiveSeqState = E_SEQ_GENERAL.DONE) 
		THEN
			eSeq := E_SEQ_CYLINDER.BASE;
		END_IF
    
  E_SEQ_CYLINDER.SET_WORK_PRESSURE_ZERO: _m_Seq_SET_WORK_PRESSURE_ZERO();
    IF TRUE
		AND (stSeqCtrlGeneral.eActiveSeqState = E_SEQ_GENERAL.DONE) 
		THEN
			eSeq := E_SEQ_CYLINDER.BASE;
		END_IF
  
  E_SEQ_CYLINDER.SET_ZERO_POS: _m_Seq_SET_ZERO_POS();
    IF TRUE
		AND (stSeqCtrlGeneral.eActiveSeqState = E_SEQ_GENERAL.DONE) 
		THEN
			eSeq := E_SEQ_CYLINDER.BASE;
		END_IF
  
  E_SEQ_CYLINDER.STOP: _m_Seq_STOP();
    IF TRUE
		AND (stSeqCtrlGeneral.eActiveSeqState = E_SEQ_GENERAL.DONE) 
		THEN
			eSeq := E_SEQ_CYLINDER.BASE;
		END_IF
    
  E_SEQ_CYLINDER.STOP_AND_LOCK: _m_Seq_STOP_AND_LOCK();
    IF TRUE
		AND (stSeqCtrlGeneral.eActiveSeqState = E_SEQ_GENERAL.DONE) 
		THEN
			eSeq := E_SEQ_CYLINDER.BASE;
		END_IF
  
  E_SEQ_CYLINDER.TO_HP: _m_Seq_TO_HP();
    IF TRUE
		AND (stSeqCtrlGeneral.eActiveSeqState = E_SEQ_GENERAL.DONE) 
		THEN
			eSeq := E_SEQ_CYLINDER.BASE;
		END_IF
  
  E_SEQ_CYLINDER.TO_SET_POS: _m_Seq_TO_SET_POS();
    IF TRUE
		AND (stSeqCtrlGeneral.eActiveSeqState = E_SEQ_GENERAL.DONE) 
		THEN
			eSeq := E_SEQ_CYLINDER.BASE;
		END_IF
  
  E_SEQ_CYLINDER.TO_WP: _m_Seq_TO_WP();
    IF TRUE
		AND (stSeqCtrlGeneral.eActiveSeqState = E_SEQ_GENERAL.DONE) 
		THEN
			eSeq := E_SEQ_CYLINDER.BASE;
		END_IF
    
  E_SEQ_CYLINDER.PRESSURE_CALIBRATION: _m_Seq_PRESSURE_CALIBRATION();
    IF TRUE
		AND (stSeqCtrlGeneral.eActiveSeqState = E_SEQ_GENERAL.DONE) 
		THEN
			eSeq := E_SEQ_CYLINDER.BASE;
		END_IF
    
  E_SEQ_CYLINDER.LOW_PRESSURE_CALIBRATION: _m_Seq_LOW_PRESSURE_CALIBRATION();
    IF TRUE
		AND (stSeqCtrlGeneral.eActiveSeqState = E_SEQ_GENERAL.DONE) 
		THEN
			eSeq := E_SEQ_CYLINDER.BASE;
		END_IF
    
  E_SEQ_CYLINDER.LOW_PRESSURE_MODE: _m_Seq_LOW_PRESSURE_MODE();
    IF TRUE
		AND (stSeqCtrlGeneral.eActiveSeqState = E_SEQ_GENERAL.DONE) 
		THEN
			eSeq := E_SEQ_CYLINDER.BASE;
		END_IF
    
  E_SEQ_CYLINDER.OPEN_RESERVOIR: _m_Seq_OPEN_RESERVOIR();
    IF TRUE
		AND (stSeqCtrlGeneral.eActiveSeqState = E_SEQ_GENERAL.DONE) 
		THEN
			eSeq := E_SEQ_CYLINDER.BASE;
		END_IF
    
  E_SEQ_CYLINDER.OPEN_LOCK_VALVES: _m_Seq_OPEN_LOCK_VALVES();
    IF TRUE
		AND (stSeqCtrlGeneral.eActiveSeqState = E_SEQ_GENERAL.DONE) 
		THEN
			eSeq := E_SEQ_CYLINDER.BASE;
		END_IF
    
  E_SEQ_CYLINDER.PUMP2_ADD: _m_Seq_PUMP2_ADD();
    IF TRUE
		AND (stSeqCtrlGeneral.eActiveSeqState = E_SEQ_GENERAL.DONE) 
		THEN
			eSeq := E_SEQ_CYLINDER.BASE;
		END_IF
    
  E_SEQ_CYLINDER.PUMP3_ADD: _m_Seq_PUMP3_ADD();
    IF TRUE
		AND (stSeqCtrlGeneral.eActiveSeqState = E_SEQ_GENERAL.DONE) 
		THEN
			eSeq := E_SEQ_CYLINDER.BASE;
		END_IF
    
  E_SEQ_CYLINDER.PUMP4_ADD: _m_Seq_PUMP4_ADD();
    IF TRUE
		AND (stSeqCtrlGeneral.eActiveSeqState = E_SEQ_GENERAL.DONE) 
		THEN
			eSeq := E_SEQ_CYLINDER.BASE;
		END_IF

  // End
	E_SEQ_CYLINDER.END:;
	E_SEQ_CYLINDER.ERROR_SEQ:;	
END_CASE

strTemp:=TO_STRING(eSeq);

METHOD PRIVATE _m_DebugManager
VAR_INPUT
	iStepID: int;
END_VAR
IF TRUE
AND THIS^.stSeqCtrlGeneral.bDebugModeActive 
AND NOT THIS^.stSeqCtrlGeneral.bActiveStep
THEN


THIS^.stSeqCtrlGeneral.bBreakpointActive:=FALSE;

FOR i:=0 TO 10 DO
	
	IF TRUE
	AND iStepID=THIS^.stSeqCtrlGeneral.listBreakpoint[i] 
	AND iStepID<>0
	THEN
		EXIT;
	END_IF
END_FOR
IF (i<=10) THEN
	THIS^.stSeqCtrlGeneral.bBreakpointActive:=TRUE;
END_IF

END_IF
END_METHOD

METHOD PRIVATE _m_Delay : BOOL
VAR_INPUT
	DelayTime:	TIME;
END_VAR
THIS^.stSeqCtrlGeneral.bDelayActive:=TRUE;
THIS^.stSeqCtrlGeneral.tDelay:=DelayTime;
_m_Delay:=FALSE;
IF THIS^.stSeqCtrlGeneral.tonDelay.Q THEN
	_m_Delay:=TRUE;
END_IF
END_METHOD

METHOD PRIVATE _m_GeneralStepSetting : BOOL
VAR_INPUT
	StepType:			    	E_STEP_STATE_TYPE;
	InfoTextID:					STRING(20);
	EnableDebug:	   			BOOL;	
	
END_VAR
IF THIS^.stSeqCtrlGeneral.bActiveStep THEN
	THIS^.stSeqCtrlGeneral.eStep_Type:=StepType;
	THIS^.stSeqCtrlGeneral.strExtraInfo:= GenLib.F_RET_TXTLIST_ENTRY(strPortNr:='851',strID:='',strTxtLstName:=InfoTextID);
END_IF
END_METHOD

METHOD PRIVATE _m_HMI : BOOL
VAR_INPUT
END_VAR
// HMI
//stHMI.bInHP := P_Position <= P_MinPosVal + 1;
//stHMI.bInWP := P_Position >= P_MaxPosVal - 1;
//stHMI.bPressureOk := P_PressureOk;
//stHMI.lrCurrentPos := P_Position;
//stHMI.lrMaxPosVal := P_MaxPosVal;
//stHMI.lrMinPosVal := P_MinPosVal;
//stHMI.lrPosToSet := lrToSetPos;
THIS^.stHMI.sState := TO_STRING(THIS^.eSeq);
//stHMI.uiSpeedInPercent
END_METHOD

METHOD PRIVATE _m_ManualOperation : BOOL
VAR_INPUT
END_VAR
IF TRUE 
AND THIS^.itfOpMode.P_OP_MODE_STATE = OP_MODE.MANUAL 
AND THIS^.itfOpModeVisu.P_HandSelected
AND THIS^.stHMI.bToHPTriggered
AND NOT THIS^.bJogCtrlBusy
THEN
  THIS^.stSeqCtrlGeneral.eActiveSeqState := E_SEQ_GENERAL.READY;
  THIS^.bStartHPTrigger := TRUE;
  THIS^.bJogCtrlBusy := TRUE;
ELSIF TRUE 
AND THIS^.itfOpMode.P_OP_MODE_STATE = OP_MODE.MANUAL 
AND THIS^.itfOpModeVisu.P_HandSelected
AND THIS^.stHMI.bToWPTriggered
AND NOT THIS^.bJogCtrlBusy
THEN
  THIS^.stSeqCtrlGeneral.eActiveSeqState := E_SEQ_GENERAL.READY;
  THIS^.bStartWPTrigger := TRUE;
  THIS^.bJogCtrlBusy := TRUE; 
ELSIF TRUE 
AND THIS^.itfOpMode.P_OP_MODE_STATE = OP_MODE.MANUAL 
AND THIS^.itfOpModeVisu.P_HandSelected
AND THIS^.stHMI.bToSetPosTriggered
AND NOT THIS^.bJogCtrlBusy
THEN
  //M_ToSetPos(lrToSetPos:= 500, rSpeedInPercent:= 100);
  THIS^.bJogCtrlBusy := TRUE;
ELSIF TRUE 
AND THIS^.itfOpMode.P_OP_MODE_STATE = OP_MODE.MANUAL 
AND THIS^.itfOpModeVisu.P_HandSelected
AND NOT THIS^.stHMI.bToHPTriggered
AND NOT THIS^.stHMI.bToWPTriggered
AND NOT THIS^.stHMI.bToSetPosTriggered
AND THIS^.bJogCtrlBusy
THEN
  THIS^.stSeqCtrlGeneral.eActiveSeqState := E_SEQ_GENERAL.READY;
  THIS^.bStopTrigger := TRUE;
  THIS^.bStartHPTrigger := FALSE;
  THIS^.bStartWPTrigger := FALSE;
  THIS^.bJogCtrlBusy := FALSE;
END_IF



IF THIS^.bStartWPTrigger THEN
  IF M_ToWP(ePressureType:= E_PRESSURE_TYPE.BAR, 
            rWorkPressure:= 10, 
            bPressureRegulation:= FALSE,
            eSpeedType:= E_SPEED_TYPE.PERCENT, 
            rSpeed:= 100) THEN
    THIS^.bStartWPTrigger := FALSE;
	END_IF
END_IF
IF THIS^.bStartHPTrigger THEN
  IF M_ToHP(ePressureType:= E_PRESSURE_TYPE.BAR, 
            rWorkPressure:= 10, 
            bPressureRegulation:= FALSE,
            eSpeedType:= E_SPEED_TYPE.PERCENT, 
            rSpeed:= 100) THEN
    THIS^.bStartHPTrigger := FALSE;
	END_IF
END_IF
IF THIS^.bStopTrigger THEN
  IF M_Stop() THEN
    THIS^.bStopTrigger := FALSE;
	END_IF
END_IF
END_METHOD

METHOD PRIVATE _m_PressureCalibration : BOOL
VAR_INPUT
END_VAR
// Calibration clicked
IF TRUE
AND THIS^.itfOpMode.P_OP_MODE_STATE = OP_MODE.MANUAL 
AND THIS^.bStartCalibrationClicked 
THEN
  IF M_PressureCalibration() THEN
    THIS^.stSeqCtrlGeneral.eActiveSeqState := E_SEQ_GENERAL.READY;
    THIS^.bStartCalibrationClicked := FALSE;
	END_IF
END_IF
IF TRUE
AND THIS^.itfOpMode.P_OP_MODE_STATE = OP_MODE.MANUAL 
AND THIS^.bStartLPCalibrationClicked 
THEN
  IF M_LowPressureCalibration() THEN
    THIS^.stSeqCtrlGeneral.eActiveSeqState := E_SEQ_GENERAL.READY;
    THIS^.bStartLPCalibrationClicked := FALSE;
	END_IF
END_IF
END_METHOD

(******************Description****************)
// This function allows variable pressure control
(*********************************************)
METHOD PRIVATE _m_PressureRegulation : BOOL
VAR_INPUT
END_VAR
IF TRUE
AND THIS^.rCurrentForceInN < THIS^.rActiveForce 
AND THIS^.iCorrectedPressureAsValue < 32768
AND THIS^.bPressureRegulationTrigger
AND NOT THIS^.bPressureRegulationBusy
THEN
  IF ABS(THIS^.rCurrentForceInN - THIS^.rActiveForce) > THIS^.rPressureRegulationTolerance THEN
    //THIS^.iCorrectedPressureAsValue := THIS^.iCorrectedPressureAsValue + 100;
    THIS^.iCorrectedPressureAsValue := TO_INT(THIS^.iCorrectedPressureAsValue + ABS((THIS^.rCurrentForceInN - THIS^.rActiveForce) * THIS^.rPressureRegulationFactor));
    THIS^.bPressureCorrectionTrigger := TRUE;
  END_IF
ELSIF TRUE
AND THIS^.rCurrentForceInN > THIS^.rActiveForce 
AND THIS^.iCorrectedPressureAsValue > 0
AND THIS^.bPressureRegulationTrigger
AND NOT THIS^.bPressureRegulationBusy
THEN
  IF ABS(THIS^.rCurrentForceInN - THIS^.rActiveForce) > THIS^.rPressureRegulationTolerance THEN
    //THIS^.iCorrectedPressureAsValue := THIS^.iCorrectedPressureAsValue - 100;
    THIS^.iCorrectedPressureAsValue := TO_INT(THIS^.iCorrectedPressureAsValue - ABS((THIS^.rCurrentForceInN - THIS^.rActiveForce) * THIS^.rPressureRegulationFactor));
    THIS^.bPressureCorrectionTrigger := TRUE;
  END_IF
END_IF

// Set Valve value correction
IF THIS^.bPressureCorrectionTrigger THEN
  THIS^.bPressureRegulationBusy:= TRUE;
  CASE THIS^.uiPressureRegulationSeq OF
    0:;
      IF THIS^.itfValve_PressureLimit.M_SetReady() THEN
        THIS^.uiPressureRegulationSeq := 1;
	    END_IF
    1:;
      IF THIS^.itfValve_PressureLimit.M_SetLimit(ePressureType:= E_PRESSURE_TYPE.VALUE, rLimit:= iCorrectedPressureAsValue) THEN
        THIS^.bPressureCorrectionTrigger := FALSE;
        THIS^.bPressureRegulationBusy := FALSE;
        THIS^.uiPressureRegulationSeq := 0;
	    END_IF
	END_CASE
END_IF
END_METHOD

METHOD PRIVATE _m_Recording : BOOL
VAR_INPUT
END_VAR
VAR
	i:                      DINT;
END_VAR
// Recording data for 5s
tonSaveInterval(IN:= NOT tonSaveInterval.Q, pt:= T#100MS);

IF iCntRecord > 499 OR iCntRecord < 0 THEN
	iCntRecord := 0;
END_IF

IF THIS^.tonSaveInterval.Q THEN
	FOR i := 299 TO 1 BY -1 DO
		THIS^.stRecord.listRecordData[i].rPosition := THIS^.stRecord.listRecordData[i - 1].rPosition;	                                  		
		THIS^.stRecord.listRecordData[i].rPressureInBar := THIS^.stRecord.listRecordData[i - 1].rPressureInBar;
	END_FOR		

	// Messergebnisse in Array eintragen	
	THIS^.stRecord.listRecordData[i].rPosition :=	THIS^.lrPos;
	THIS^.stRecord.listRecordData[i].rPressureInBar := THIS^.rCurrentPressureInBar;
END_IF

// Calibration table
FOR THIS^.iii := 1 TO 7 BY 1 DO
  THIS^.listCylCalibration[2, THIS^.iii] := TO_LREAL(THIS^.listCalibrationTable[iii].uiValue);
  THIS^.listCylCalibration[1, THIS^.iii] := TO_LREAL(THIS^.listCalibrationTable[iii].uiPressure);
  THIS^.listLPCylCalibration[2, THIS^.iii] := TO_LREAL(THIS^.listLPCalibrationTable[iii].uiValue);
  THIS^.listLPCylCalibration[1, THIS^.iii] := TO_LREAL(THIS^.listLPCalibrationTable[iii].uiPressure);
END_FOR

// Position
THIS^.lrPos := -(THIS^.lrCurrentPosAbs / 1000 - THIS^.lrPosZero);
THIS^.rStrokeLength := -(THIS^.lrPosMax - THIS^.lrPosZero);

// Speed
IF THIS^.x < 1 OR THIS^.x > 100 THEN
  THIS^.x := 1;
END_IF
THIS^.listPosTable[THIS^.x] := THIS^.lrPos - THIS^.lrLastPos;
THIS^.lrTotalPath := 0;
FOR THIS^.xx := 1 TO 100 BY 1 DO
  THIS^.lrTotalPath := THIS^.lrTotalPath + THIS^.listPosTable[THIS^.xx];
END_FOR
THIS^.rCurrentSpeedInMmPerS := THIS^.lrTotalPath;
THIS^.x := THIS^.x + 1;
THIS^.lrLastPos := THIS^.lrPos;
END_METHOD

METHOD PRIVATE _m_SaveLastStep : BOOL
VAR_INPUT
END_VAR
VAR
	i: dint;
END_VAR
IF NOT THIS^.stSeqCtrlGeneral.bActiveStep THEN
	
	FOR i:=49 TO 1 BY -1 DO
			stSeqCtrlGeneral.listLastSteps[i].strStepName:=stSeqCtrlGeneral.listLastSteps[i-1].strStepName;
			stSeqCtrlGeneral.listLastSteps[i].tStepTime:=stSeqCtrlGeneral.listLastSteps[i-1].tStepTime;
			stSeqCtrlGeneral.listLastSteps[i].tDelayTime:=stSeqCtrlGeneral.listLastSteps[i-1].tDelayTime;
	END_FOR
	stSeqCtrlGeneral.listLastSteps[0].strStepName:=TO_STRING(THIS^.eSeq);
	stSeqCtrlGeneral.listLastSteps[1].tStepTime:=THIS^.stSeqCtrlGeneral.tonStepTime.ET;
	stSeqCtrlGeneral.listLastSteps[1].tStepTime:=THIS^.stSeqCtrlGeneral.tonDelay.ET;
ELSE
	stSeqCtrlGeneral.listLastSteps[0].tStepTime:=THIS^.stSeqCtrlGeneral.tonStepTime.ET;
	stSeqCtrlGeneral.listLastSteps[0].tDelayTime:=THIS^.stSeqCtrlGeneral.tonDelay.ET;	
END_IF
END_METHOD

METHOD PRIVATE _m_Seq_INIT : E_SEQ_PROCESS
VAR_INPUT
END_VAR
VAR
	ActiveSeq: STRING;
END_VAR
VAR
	
END_VAR
//THIS^._m_GeneralStepSetting(StepType:=E_STEP_STATE_TYPE.INIT,
ActiveSeq := TO_STRING(THIS^.eSeq);

CASE THIS^.stSeqCtrlGeneral.eActiveSeqState OF
E_SEQ_GENERAL.READY:;

	
E_SEQ_GENERAL.EXECUTE:;
	IF TRUE
	THEN
		THIS^.stSeqCtrlGeneral.eActiveSeqState := E_SEQ_GENERAL.RESET;
	END_IF
E_SEQ_GENERAL.RESET:;
	stSeqCtrlGeneral.iInternalSeqStateCase := 0;
	IF TRUE
	THEN
    THIS^.bRegulation := FALSE;
		THIS^.stSeqCtrlGeneral.eActiveSeqState := E_SEQ_GENERAL.BUSY;
	END_IF
  
E_SEQ_GENERAL.BUSY:;
	CASE THIS^.stSeqCtrlGeneral.iInternalSeqStateCase OF
		0:	// Reset valves
      IF TRUE
      AND THIS^.itfValve_CylCtrl.M_Reset()
      AND THIS^.itfValve_LockA.M_ToHP(tDelay:= T#10MS)
      AND THIS^.itfValve_LockB.M_ToHP(tDelay:= T#10MS)
      AND THIS^.itfValve_AddPump2.M_ToHP(tDelay:= T#10MS)
      AND THIS^.itfValve_AddPump3.M_ToHP(tDelay:= T#10MS)
      AND THIS^.itfValve_AddPump4.M_ToHP(tDelay:= T#10MS)
      AND THIS^.itfValve_PressureReservoirAAdd.M_ToHP(tDelay:= T#10MS)
      AND THIS^.itfValve_PressureReservoirBAdd.M_ToHP(tDelay:= T#10MS)
      AND THIS^.itfValve_SensorBreakPressureAAdd.M_ToHP(tDelay:= T#10MS)
      AND THIS^.itfValve_SensorBreakPressureBAdd.M_ToHP(tDelay:= T#10MS)
      AND THIS^.itfShutOffValve_LowPressure.M_Close()
			THEN 
				THIS^.stSeqCtrlGeneral.iInternalSeqStateCase := 1000;
			END_IF
      
    1000: // Exit step
      IF TRUE
			THEN 
				THIS^.stSeqCtrlGeneral.iInternalSeqStateCase := 9999;
			END_IF
      
	ELSE
		THIS^.stSeqCtrlGeneral.eActiveSeqState := E_SEQ_GENERAL.DONE;  
	END_CASE
	THIS^.stSeqCtrlGeneral.strExtraInfo := CONCAT('Internal state: ', TO_STRING(THIS^.stSeqCtrlGeneral.iInternalSeqStateCase));
  
E_SEQ_GENERAL.DONE:;
E_SEQ_GENERAL.ERROR:;
E_SEQ_GENERAL.TIME_OUT:; 

